(* Logix 5000 project; controller reports 1756-L63 rev 20.11; software revision 20.04; part 19 of 52 *)

        [1096].log_data[14].valid := 1, [1096].log_data[15].valid := 1, [1096].log_data[16].valid := 1, [1096].log_data[17].valid := 1, [1096].log_data[18].valid := 1, [1096].log_data[19].valid := 1, [1096].time.Year := 2023, [1096].time.Month := 1, [1096].time.Day := 13, [1096].time.Hour := 11, [1096].time.Minute := 44, [1096].time.Second := 59, [1097].log_data[0].min := 1.0, [1097].log_data[0].max := 1.0, [1097].log_data[0].total := 300.0, [1097].log_data[0].time := 300.0, [1097].log_data[0].minminute := 45, [1097].log_data[0].maxminute := 45, [1097].log_data[0].valid := 1, [1097].log_data[1].valid := 1, [1097].log_data[2].valid := 1, [1097].log_data[3].valid := 1, [1097].log_data[4].valid := 1, [1097].log_data[5].valid := 1, [1097].log_data[6].valid := 1, [1097].log_data[7].valid := 1, [1097].log_data[8].valid := 1, [1097].log_data[9].valid := 1, [1097].log_data[10].valid := 1, [1097].log_data[11].valid := 1, [1097].log_data[12].valid := 1, [1097].log_data[13].valid := 1, [1097].log_data[14].valid := 1, [1097].log_data[15].valid := 1, [1097].log_data[16].valid := 1, [1097].log_data[17].valid := 1, [1097].log_data[18].valid := 1, [1097].log_data[19].valid := 1, [1097].time.Year := 2023, [1097].time.Month := 1, [1097].time.Day := 13, [1097].time.Hour := 11, [1097].time.Minute := 49, [1097].time.Second := 59, [1098].log_data[0].min := 1.0, [1098].log_data[0].max := 1.0, [1098].log_data[0].total := 300.0, [1098].log_data[0].time := 300.0, [1098].log_data[0].minminute := 50, [1098].log_data[0].maxminute := 50, [1098].log_data[0].valid := 1, [1098].log_data[1].valid := 1, [1098].log_data[2].valid := 1, [1098].log_data[3].valid := 1, [1098].log_data[4].valid := 1, [1098].log_data[5].valid := 1, [1098].log_data[6].valid := 1, [1098].log_data[7].valid := 1, [1098].log_data[8].valid := 1, [1098].log_data[9].valid := 1,
        [1098].log_data[10].valid := 1, [1098].log_data[11].valid := 1, [1098].log_data[12].valid := 1, [1098].log_data[13].valid := 1, [1098].log_data[14].valid := 1, [1098].log_data[15].valid := 1, [1098].log_data[16].valid := 1, [1098].log_data[17].valid := 1, [1098].log_data[18].valid := 1, [1098].log_data[19].valid := 1, [1098].time.Year := 2023, [1098].time.Month := 1, [1098].time.Day := 13, [1098].time.Hour := 11, [1098].time.Minute := 54, [1098].time.Second := 59, [1099].log_data[0].min := 1.0, [1099].log_data[0].max := 1.0, [1099].log_data[0].total := 300.0, [1099].log_data[0].time := 300.0, [1099].log_data[0].minminute := 55, [1099].log_data[0].maxminute := 55, [1099].log_data[0].valid := 1, [1099].log_data[1].valid := 1, [1099].log_data[2].valid := 1, [1099].log_data[3].valid := 1, [1099].log_data[4].valid := 1, [1099].log_data[5].valid := 1, [1099].log_data[6].valid := 1, [1099].log_data[7].valid := 1, [1099].log_data[8].valid := 1, [1099].log_data[9].valid := 1, [1099].log_data[10].valid := 1, [1099].log_data[11].valid := 1, [1099].log_data[12].valid := 1, [1099].log_data[13].valid := 1, [1099].log_data[14].valid := 1, [1099].log_data[15].valid := 1, [1099].log_data[16].valid := 1, [1099].log_data[17].valid := 1, [1099].log_data[18].valid := 1, [1099].log_data[19].valid := 1, [1099].time.Year := 2023, [1099].time.Month := 1, [1099].time.Day := 13, [1099].time.Hour := 11, [1099].time.Minute := 59, [1099].time.Second := 59, [1100].log_data[0].min := 1.0, [1100].log_data[0].max := 1.0, [1100].log_data[0].total := 300.0, [1100].log_data[0].time := 300.0, [1100].log_data[0].valid := 1, [1100].log_data[1].valid := 1, [1100].log_data[2].valid := 1, [1100].log_data[3].valid := 1, [1100].log_data[4].valid := 1, [1100].log_data[5].valid := 1, [1100].log_data[6].valid := 1, [1100].log_data[7].valid := 1,
        [1100].log_data[8].valid := 1, [1100].log_data[9].valid := 1, [1100].log_data[10].valid := 1, [1100].log_data[11].valid := 1, [1100].log_data[12].valid := 1, [1100].log_data[13].valid := 1, [1100].log_data[14].valid := 1, [1100].log_data[15].valid := 1, [1100].log_data[16].valid := 1, [1100].log_data[17].valid := 1, [1100].log_data[18].valid := 1, [1100].log_data[19].valid := 1, [1100].time.Year := 2023, [1100].time.Month := 1, [1100].time.Day := 13, [1100].time.Hour := 12, [1100].time.Minute := 4, [1100].time.Second := 59, [1101].log_data[0].min := 1.0, [1101].log_data[0].max := 1.0, [1101].log_data[0].total := 300.0, [1101].log_data[0].time := 300.0, [1101].log_data[0].minminute := 5, [1101].log_data[0].maxminute := 5, [1101].log_data[0].valid := 1, [1101].log_data[1].valid := 1, [1101].log_data[2].valid := 1, [1101].log_data[3].valid := 1, [1101].log_data[4].valid := 1, [1101].log_data[5].valid := 1, [1101].log_data[6].valid := 1, [1101].log_data[7].valid := 1, [1101].log_data[8].valid := 1, [1101].log_data[9].valid := 1, [1101].log_data[10].valid := 1, [1101].log_data[11].valid := 1, [1101].log_data[12].valid := 1, [1101].log_data[13].valid := 1, [1101].log_data[14].valid := 1, [1101].log_data[15].valid := 1, [1101].log_data[16].valid := 1, [1101].log_data[17].valid := 1, [1101].log_data[18].valid := 1, [1101].log_data[19].valid := 1, [1101].time.Year := 2023, [1101].time.Month := 1, [1101].time.Day := 13, [1101].time.Hour := 12, [1101].time.Minute := 9, [1101].time.Second := 59, [1102].log_data[0].min := 1.0, [1102].log_data[0].max := 1.0, [1102].log_data[0].total := 300.0, [1102].log_data[0].time := 300.0, [1102].log_data[0].minminute := 10, [1102].log_data[0].maxminute := 10, [1102].log_data[0].valid := 1, [1102].log_data[1].valid := 1, [1102].log_data[2].valid := 1, [1102].log_data[3].valid := 1,
        [1102].log_data[4].valid := 1, [1102].log_data[5].valid := 1, [1102].log_data[6].valid := 1, [1102].log_data[7].valid := 1, [1102].log_data[8].valid := 1, [1102].log_data[9].valid := 1, [1102].log_data[10].valid := 1, [1102].log_data[11].valid := 1, [1102].log_data[12].valid := 1, [1102].log_data[13].valid := 1, [1102].log_data[14].valid := 1, [1102].log_data[15].valid := 1, [1102].log_data[16].valid := 1, [1102].log_data[17].valid := 1, [1102].log_data[18].valid := 1, [1102].log_data[19].valid := 1, [1102].time.Year := 2023, [1102].time.Month := 1, [1102].time.Day := 13, [1102].time.Hour := 12, [1102].time.Minute := 14, [1102].time.Second := 59, [1103].log_data[0].min := 1.0, [1103].log_data[0].max := 1.0, [1103].log_data[0].total := 300.0, [1103].log_data[0].time := 300.0, [1103].log_data[0].minminute := 15, [1103].log_data[0].maxminute := 15, [1103].log_data[0].valid := 1, [1103].log_data[1].valid := 1, [1103].log_data[2].valid := 1, [1103].log_data[3].valid := 1, [1103].log_data[4].valid := 1, [1103].log_data[5].valid := 1, [1103].log_data[6].valid := 1, [1103].log_data[7].valid := 1, [1103].log_data[8].valid := 1, [1103].log_data[9].valid := 1, [1103].log_data[10].valid := 1, [1103].log_data[11].valid := 1, [1103].log_data[12].valid := 1, [1103].log_data[13].valid := 1, [1103].log_data[14].valid := 1, [1103].log_data[15].valid := 1, [1103].log_data[16].valid := 1, [1103].log_data[17].valid := 1, [1103].log_data[18].valid := 1, [1103].log_data[19].valid := 1, [1103].time.Year := 2023, [1103].time.Month := 1, [1103].time.Day := 13, [1103].time.Hour := 12, [1103].time.Minute := 19, [1103].time.Second := 59, [1104].log_data[0].min := 1.0, [1104].log_data[0].max := 1.0, [1104].log_data[0].total := 300.0, [1104].log_data[0].time := 300.0, [1104].log_data[0].minminute := 20, [1104].log_data[0].maxminute := 20,
        [1104].log_data[0].valid := 1, [1104].log_data[1].valid := 1, [1104].log_data[2].valid := 1, [1104].log_data[3].valid := 1, [1104].log_data[4].valid := 1, [1104].log_data[5].valid := 1, [1104].log_data[6].valid := 1, [1104].log_data[7].valid := 1, [1104].log_data[8].valid := 1, [1104].log_data[9].valid := 1, [1104].log_data[10].valid := 1, [1104].log_data[11].valid := 1, [1104].log_data[12].valid := 1, [1104].log_data[13].valid := 1, [1104].log_data[14].valid := 1, [1104].log_data[15].valid := 1, [1104].log_data[16].valid := 1, [1104].log_data[17].valid := 1, [1104].log_data[18].valid := 1, [1104].log_data[19].valid := 1, [1104].time.Year := 2023, [1104].time.Month := 1, [1104].time.Day := 13, [1104].time.Hour := 12, [1104].time.Minute := 24, [1104].time.Second := 59, [1105].log_data[0].min := 1.0, [1105].log_data[0].max := 1.0, [1105].log_data[0].total := 300.0, [1105].log_data[0].time := 300.0, [1105].log_data[0].minminute := 25, [1105].log_data[0].maxminute := 25, [1105].log_data[0].valid := 1, [1105].log_data[1].valid := 1, [1105].log_data[2].valid := 1, [1105].log_data[3].valid := 1, [1105].log_data[4].valid := 1, [1105].log_data[5].valid := 1, [1105].log_data[6].valid := 1, [1105].log_data[7].valid := 1, [1105].log_data[8].valid := 1, [1105].log_data[9].valid := 1, [1105].log_data[10].valid := 1, [1105].log_data[11].valid := 1, [1105].log_data[12].valid := 1, [1105].log_data[13].valid := 1, [1105].log_data[14].valid := 1, [1105].log_data[15].valid := 1, [1105].log_data[16].valid := 1, [1105].log_data[17].valid := 1, [1105].log_data[18].valid := 1, [1105].log_data[19].valid := 1, [1105].time.Year := 2023, [1105].time.Month := 1, [1105].time.Day := 13, [1105].time.Hour := 12, [1105].time.Minute := 29, [1105].time.Second := 59, [1106].log_data[0].min := 1.0, [1106].log_data[0].max := 1.0,
        [1106].log_data[0].total := 300.0, [1106].log_data[0].time := 300.0, [1106].log_data[0].minminute := 30, [1106].log_data[0].maxminute := 30, [1106].log_data[0].valid := 1, [1106].log_data[1].valid := 1, [1106].log_data[2].valid := 1, [1106].log_data[3].valid := 1, [1106].log_data[4].valid := 1, [1106].log_data[5].valid := 1, [1106].log_data[6].valid := 1, [1106].log_data[7].valid := 1, [1106].log_data[8].valid := 1, [1106].log_data[9].valid := 1, [1106].log_data[10].valid := 1, [1106].log_data[11].valid := 1, [1106].log_data[12].valid := 1, [1106].log_data[13].valid := 1, [1106].log_data[14].valid := 1, [1106].log_data[15].valid := 1, [1106].log_data[16].valid := 1, [1106].log_data[17].valid := 1, [1106].log_data[18].valid := 1, [1106].log_data[19].valid := 1, [1106].time.Year := 2023, [1106].time.Month := 1, [1106].time.Day := 13, [1106].time.Hour := 12, [1106].time.Minute := 34, [1106].time.Second := 59, [1107].log_data[0].min := 1.0, [1107].log_data[0].max := 1.0, [1107].log_data[0].total := 300.0, [1107].log_data[0].time := 300.0, [1107].log_data[0].minminute := 35, [1107].log_data[0].maxminute := 35, [1107].log_data[0].valid := 1, [1107].log_data[1].valid := 1, [1107].log_data[2].valid := 1, [1107].log_data[3].valid := 1, [1107].log_data[4].valid := 1, [1107].log_data[5].valid := 1, [1107].log_data[6].valid := 1, [1107].log_data[7].valid := 1, [1107].log_data[8].valid := 1, [1107].log_data[9].valid := 1, [1107].log_data[10].valid := 1, [1107].log_data[11].valid := 1, [1107].log_data[12].valid := 1, [1107].log_data[13].valid := 1, [1107].log_data[14].valid := 1, [1107].log_data[15].valid := 1, [1107].log_data[16].valid := 1, [1107].log_data[17].valid := 1, [1107].log_data[18].valid := 1, [1107].log_data[19].valid := 1, [1107].time.Year := 2023, [1107].time.Month := 1, [1107].time.Day := 13, [1107].time.Hour := 12,
        [1107].time.Minute := 39, [1107].time.Second := 59, [1108].log_data[0].min := 1.0, [1108].log_data[0].max := 1.0, [1108].log_data[0].total := 300.0, [1108].log_data[0].time := 300.0, [1108].log_data[0].minminute := 40, [1108].log_data[0].maxminute := 40, [1108].log_data[0].valid := 1, [1108].log_data[1].valid := 1, [1108].log_data[2].valid := 1, [1108].log_data[3].valid := 1, [1108].log_data[4].valid := 1, [1108].log_data[5].valid := 1, [1108].log_data[6].valid := 1, [1108].log_data[7].valid := 1, [1108].log_data[8].valid := 1, [1108].log_data[9].valid := 1, [1108].log_data[10].valid := 1, [1108].log_data[11].valid := 1, [1108].log_data[12].valid := 1, [1108].log_data[13].valid := 1, [1108].log_data[14].valid := 1, [1108].log_data[15].valid := 1, [1108].log_data[16].valid := 1, [1108].log_data[17].valid := 1, [1108].log_data[18].valid := 1, [1108].log_data[19].valid := 1, [1108].time.Year := 2023, [1108].time.Month := 1, [1108].time.Day := 13, [1108].time.Hour := 12, [1108].time.Minute := 44, [1108].time.Second := 59, [1109].log_data[0].min := 1.0, [1109].log_data[0].max := 1.0, [1109].log_data[0].total := 300.0, [1109].log_data[0].time := 300.0, [1109].log_data[0].minminute := 45, [1109].log_data[0].maxminute := 45, [1109].log_data[0].valid := 1, [1109].log_data[1].valid := 1, [1109].log_data[2].valid := 1, [1109].log_data[3].valid := 1, [1109].log_data[4].valid := 1, [1109].log_data[5].valid := 1, [1109].log_data[6].valid := 1, [1109].log_data[7].valid := 1, [1109].log_data[8].valid := 1, [1109].log_data[9].valid := 1, [1109].log_data[10].valid := 1, [1109].log_data[11].valid := 1, [1109].log_data[12].valid := 1, [1109].log_data[13].valid := 1, [1109].log_data[14].valid := 1, [1109].log_data[15].valid := 1, [1109].log_data[16].valid := 1, [1109].log_data[17].valid := 1, [1109].log_data[18].valid := 1, [1109].log_data[19].valid := 1,
        [1109].time.Year := 2023, [1109].time.Month := 1, [1109].time.Day := 13, [1109].time.Hour := 12, [1109].time.Minute := 49, [1109].time.Second := 59, [1110].log_data[0].min := 1.0, [1110].log_data[0].max := 1.0, [1110].log_data[0].total := 300.0, [1110].log_data[0].time := 300.0, [1110].log_data[0].minminute := 50, [1110].log_data[0].maxminute := 50, [1110].log_data[0].valid := 1, [1110].log_data[1].valid := 1, [1110].log_data[2].valid := 1, [1110].log_data[3].valid := 1, [1110].log_data[4].valid := 1, [1110].log_data[5].valid := 1, [1110].log_data[6].valid := 1, [1110].log_data[7].valid := 1, [1110].log_data[8].valid := 1, [1110].log_data[9].valid := 1, [1110].log_data[10].valid := 1, [1110].log_data[11].valid := 1, [1110].log_data[12].valid := 1, [1110].log_data[13].valid := 1, [1110].log_data[14].valid := 1, [1110].log_data[15].valid := 1, [1110].log_data[16].valid := 1, [1110].log_data[17].valid := 1, [1110].log_data[18].valid := 1, [1110].log_data[19].valid := 1, [1110].time.Year := 2023, [1110].time.Month := 1, [1110].time.Day := 13, [1110].time.Hour := 12, [1110].time.Minute := 54, [1110].time.Second := 59, [1111].log_data[0].min := 1.0, [1111].log_data[0].max := 1.0, [1111].log_data[0].total := 300.0, [1111].log_data[0].time := 300.0, [1111].log_data[0].minminute := 55, [1111].log_data[0].maxminute := 55, [1111].log_data[0].valid := 1, [1111].log_data[1].valid := 1, [1111].log_data[2].valid := 1, [1111].log_data[3].valid := 1, [1111].log_data[4].valid := 1, [1111].log_data[5].valid := 1, [1111].log_data[6].valid := 1, [1111].log_data[7].valid := 1, [1111].log_data[8].valid := 1, [1111].log_data[9].valid := 1, [1111].log_data[10].valid := 1, [1111].log_data[11].valid := 1, [1111].log_data[12].valid := 1, [1111].log_data[13].valid := 1, [1111].log_data[14].valid := 1, [1111].log_data[15].valid := 1,
        [1111].log_data[16].valid := 1, [1111].log_data[17].valid := 1, [1111].log_data[18].valid := 1, [1111].log_data[19].valid := 1, [1111].time.Year := 2023, [1111].time.Month := 1, [1111].time.Day := 13, [1111].time.Hour := 12, [1111].time.Minute := 59, [1111].time.Second := 59, [1112].log_data[0].min := 1.0, [1112].log_data[0].max := 1.0, [1112].log_data[0].total := 299.5, [1112].log_data[0].time := 299.5, [1112].log_data[0].valid := 1, [1112].log_data[1].valid := 1, [1112].log_data[2].valid := 1, [1112].log_data[3].valid := 1, [1112].log_data[4].valid := 1, [1112].log_data[5].valid := 1, [1112].log_data[6].valid := 1, [1112].log_data[7].valid := 1, [1112].log_data[8].valid := 1, [1112].log_data[9].valid := 1, [1112].log_data[10].valid := 1, [1112].log_data[11].valid := 1, [1112].log_data[12].valid := 1, [1112].log_data[13].valid := 1, [1112].log_data[14].valid := 1, [1112].log_data[15].valid := 1, [1112].log_data[16].valid := 1, [1112].log_data[17].valid := 1, [1112].log_data[18].valid := 1, [1112].log_data[19].valid := 1, [1112].time.Year := 2023, [1112].time.Month := 1, [1112].time.Day := 13, [1112].time.Hour := 13, [1112].time.Minute := 4, [1112].time.Second := 59, [1113].log_data[0].min := 1.0, [1113].log_data[0].max := 1.0, [1113].log_data[0].total := 300.0, [1113].log_data[0].time := 300.0, [1113].log_data[0].minminute := 5, [1113].log_data[0].maxminute := 5, [1113].log_data[0].valid := 1, [1113].log_data[1].valid := 1, [1113].log_data[2].valid := 1, [1113].log_data[3].valid := 1, [1113].log_data[4].valid := 1, [1113].log_data[5].valid := 1, [1113].log_data[6].valid := 1, [1113].log_data[7].valid := 1, [1113].log_data[8].valid := 1, [1113].log_data[9].valid := 1, [1113].log_data[10].valid := 1, [1113].log_data[11].valid := 1, [1113].log_data[12].valid := 1, [1113].log_data[13].valid := 1,
        [1113].log_data[14].valid := 1, [1113].log_data[15].valid := 1, [1113].log_data[16].valid := 1, [1113].log_data[17].valid := 1, [1113].log_data[18].valid := 1, [1113].log_data[19].valid := 1, [1113].time.Year := 2023, [1113].time.Month := 1, [1113].time.Day := 13, [1113].time.Hour := 13, [1113].time.Minute := 9, [1113].time.Second := 59, [1114].log_data[0].min := 1.0, [1114].log_data[0].max := 1.0, [1114].log_data[0].total := 300.0, [1114].log_data[0].time := 300.0, [1114].log_data[0].minminute := 10, [1114].log_data[0].maxminute := 10, [1114].log_data[0].valid := 1, [1114].log_data[1].valid := 1, [1114].log_data[2].valid := 1, [1114].log_data[3].valid := 1, [1114].log_data[4].valid := 1, [1114].log_data[5].valid := 1, [1114].log_data[6].valid := 1, [1114].log_data[7].valid := 1, [1114].log_data[8].valid := 1, [1114].log_data[9].valid := 1, [1114].log_data[10].valid := 1, [1114].log_data[11].valid := 1, [1114].log_data[12].valid := 1, [1114].log_data[13].valid := 1, [1114].log_data[14].valid := 1, [1114].log_data[15].valid := 1, [1114].log_data[16].valid := 1, [1114].log_data[17].valid := 1, [1114].log_data[18].valid := 1, [1114].log_data[19].valid := 1, [1114].time.Year := 2023, [1114].time.Month := 1, [1114].time.Day := 13, [1114].time.Hour := 13, [1114].time.Minute := 14, [1114].time.Second := 59, [1115].log_data[0].min := 1.0, [1115].log_data[0].max := 1.0, [1115].log_data[0].total := 300.0, [1115].log_data[0].time := 300.0, [1115].log_data[0].minminute := 15, [1115].log_data[0].maxminute := 15, [1115].log_data[0].valid := 1, [1115].log_data[1].valid := 1, [1115].log_data[2].valid := 1, [1115].log_data[3].valid := 1, [1115].log_data[4].valid := 1, [1115].log_data[5].valid := 1, [1115].log_data[6].valid := 1, [1115].log_data[7].valid := 1, [1115].log_data[8].valid := 1, [1115].log_data[9].valid := 1,
        [1115].log_data[10].valid := 1, [1115].log_data[11].valid := 1, [1115].log_data[12].valid := 1, [1115].log_data[13].valid := 1, [1115].log_data[14].valid := 1, [1115].log_data[15].valid := 1, [1115].log_data[16].valid := 1, [1115].log_data[17].valid := 1, [1115].log_data[18].valid := 1, [1115].log_data[19].valid := 1, [1115].time.Year := 2023, [1115].time.Month := 1, [1115].time.Day := 13, [1115].time.Hour := 13, [1115].time.Minute := 19, [1115].time.Second := 59, [1116].log_data[0].min := 1.0, [1116].log_data[0].max := 1.0, [1116].log_data[0].total := 300.0, [1116].log_data[0].time := 300.0, [1116].log_data[0].minminute := 20, [1116].log_data[0].maxminute := 20, [1116].log_data[0].valid := 1, [1116].log_data[1].valid := 1, [1116].log_data[2].valid := 1, [1116].log_data[3].valid := 1, [1116].log_data[4].valid := 1, [1116].log_data[5].valid := 1, [1116].log_data[6].valid := 1, [1116].log_data[7].valid := 1, [1116].log_data[8].valid := 1, [1116].log_data[9].valid := 1, [1116].log_data[10].valid := 1, [1116].log_data[11].valid := 1, [1116].log_data[12].valid := 1, [1116].log_data[13].valid := 1, [1116].log_data[14].valid := 1, [1116].log_data[15].valid := 1, [1116].log_data[16].valid := 1, [1116].log_data[17].valid := 1, [1116].log_data[18].valid := 1, [1116].log_data[19].valid := 1, [1116].time.Year := 2023, [1116].time.Month := 1, [1116].time.Day := 13, [1116].time.Hour := 13, [1116].time.Minute := 24, [1116].time.Second := 59, [1117].log_data[0].min := 1.0, [1117].log_data[0].max := 1.0, [1117].log_data[0].total := 300.0, [1117].log_data[0].time := 300.0, [1117].log_data[0].minminute := 25, [1117].log_data[0].maxminute := 25, [1117].log_data[0].valid := 1, [1117].log_data[1].valid := 1, [1117].log_data[2].valid := 1, [1117].log_data[3].valid := 1, [1117].log_data[4].valid := 1, [1117].log_data[5].valid := 1,
        [1117].log_data[6].valid := 1, [1117].log_data[7].valid := 1, [1117].log_data[8].valid := 1, [1117].log_data[9].valid := 1, [1117].log_data[10].valid := 1, [1117].log_data[11].valid := 1, [1117].log_data[12].valid := 1, [1117].log_data[13].valid := 1, [1117].log_data[14].valid := 1, [1117].log_data[15].valid := 1, [1117].log_data[16].valid := 1, [1117].log_data[17].valid := 1, [1117].log_data[18].valid := 1, [1117].log_data[19].valid := 1, [1117].time.Year := 2023, [1117].time.Month := 1, [1117].time.Day := 13, [1117].time.Hour := 13, [1117].time.Minute := 29, [1117].time.Second := 59, [1118].log_data[0].min := 1.0, [1118].log_data[0].max := 1.0, [1118].log_data[0].total := 300.0, [1118].log_data[0].time := 300.0, [1118].log_data[0].minminute := 30, [1118].log_data[0].maxminute := 30, [1118].log_data[0].valid := 1, [1118].log_data[1].valid := 1, [1118].log_data[2].valid := 1, [1118].log_data[3].valid := 1, [1118].log_data[4].valid := 1, [1118].log_data[5].valid := 1, [1118].log_data[6].valid := 1, [1118].log_data[7].valid := 1, [1118].log_data[8].valid := 1, [1118].log_data[9].valid := 1, [1118].log_data[10].valid := 1, [1118].log_data[11].valid := 1, [1118].log_data[12].valid := 1, [1118].log_data[13].valid := 1, [1118].log_data[14].valid := 1, [1118].log_data[15].valid := 1, [1118].log_data[16].valid := 1, [1118].log_data[17].valid := 1, [1118].log_data[18].valid := 1, [1118].log_data[19].valid := 1, [1118].time.Year := 2023, [1118].time.Month := 1, [1118].time.Day := 13, [1118].time.Hour := 13, [1118].time.Minute := 34, [1118].time.Second := 59, [1119].log_data[0].min := 1.0, [1119].log_data[0].max := 1.0, [1119].log_data[0].total := 300.0, [1119].log_data[0].time := 300.0, [1119].log_data[0].minminute := 35, [1119].log_data[0].maxminute := 35, [1119].log_data[0].valid := 1, [1119].log_data[1].valid := 1,
        [1119].log_data[2].valid := 1, [1119].log_data[3].valid := 1, [1119].log_data[4].valid := 1, [1119].log_data[5].valid := 1, [1119].log_data[6].valid := 1, [1119].log_data[7].valid := 1, [1119].log_data[8].valid := 1, [1119].log_data[9].valid := 1, [1119].log_data[10].valid := 1, [1119].log_data[11].valid := 1, [1119].log_data[12].valid := 1, [1119].log_data[13].valid := 1, [1119].log_data[14].valid := 1, [1119].log_data[15].valid := 1, [1119].log_data[16].valid := 1, [1119].log_data[17].valid := 1, [1119].log_data[18].valid := 1, [1119].log_data[19].valid := 1, [1119].time.Year := 2023, [1119].time.Month := 1, [1119].time.Day := 13, [1119].time.Hour := 13, [1119].time.Minute := 39, [1119].time.Second := 59, [1120].log_data[0].min := 1.0, [1120].log_data[0].max := 1.0, [1120].log_data[0].total := 300.0, [1120].log_data[0].time := 300.0, [1120].log_data[0].minminute := 40, [1120].log_data[0].maxminute := 40, [1120].log_data[0].valid := 1, [1120].log_data[1].valid := 1, [1120].log_data[2].valid := 1, [1120].log_data[3].valid := 1, [1120].log_data[4].valid := 1, [1120].log_data[5].valid := 1, [1120].log_data[6].valid := 1, [1120].log_data[7].valid := 1, [1120].log_data[8].valid := 1, [1120].log_data[9].valid := 1, [1120].log_data[10].valid := 1, [1120].log_data[11].valid := 1, [1120].log_data[12].valid := 1, [1120].log_data[13].valid := 1, [1120].log_data[14].valid := 1, [1120].log_data[15].valid := 1, [1120].log_data[16].valid := 1, [1120].log_data[17].valid := 1, [1120].log_data[18].valid := 1, [1120].log_data[19].valid := 1, [1120].time.Year := 2023, [1120].time.Month := 1, [1120].time.Day := 13, [1120].time.Hour := 13, [1120].time.Minute := 44, [1120].time.Second := 59, [1121].log_data[0].min := 1.0, [1121].log_data[0].max := 1.0, [1121].log_data[0].total := 300.0, [1121].log_data[0].time := 300.0,
        [1121].log_data[0].minminute := 45, [1121].log_data[0].maxminute := 45, [1121].log_data[0].valid := 1, [1121].log_data[1].valid := 1, [1121].log_data[2].valid := 1, [1121].log_data[3].valid := 1, [1121].log_data[4].valid := 1, [1121].log_data[5].valid := 1, [1121].log_data[6].valid := 1, [1121].log_data[7].valid := 1, [1121].log_data[8].valid := 1, [1121].log_data[9].valid := 1, [1121].log_data[10].valid := 1, [1121].log_data[11].valid := 1, [1121].log_data[12].valid := 1, [1121].log_data[13].valid := 1, [1121].log_data[14].valid := 1, [1121].log_data[15].valid := 1, [1121].log_data[16].valid := 1, [1121].log_data[17].valid := 1, [1121].log_data[18].valid := 1, [1121].log_data[19].valid := 1, [1121].time.Year := 2023, [1121].time.Month := 1, [1121].time.Day := 13, [1121].time.Hour := 13, [1121].time.Minute := 49, [1121].time.Second := 59, [1122].log_data[0].min := 1.0, [1122].log_data[0].max := 1.0, [1122].log_data[0].total := 300.0, [1122].log_data[0].time := 300.0, [1122].log_data[0].minminute := 50, [1122].log_data[0].maxminute := 50, [1122].log_data[0].valid := 1, [1122].log_data[1].valid := 1, [1122].log_data[2].valid := 1, [1122].log_data[3].valid := 1, [1122].log_data[4].valid := 1, [1122].log_data[5].valid := 1, [1122].log_data[6].valid := 1, [1122].log_data[7].valid := 1, [1122].log_data[8].valid := 1, [1122].log_data[9].valid := 1, [1122].log_data[10].valid := 1, [1122].log_data[11].valid := 1, [1122].log_data[12].valid := 1, [1122].log_data[13].valid := 1, [1122].log_data[14].valid := 1, [1122].log_data[15].valid := 1, [1122].log_data[16].valid := 1, [1122].log_data[17].valid := 1, [1122].log_data[18].valid := 1, [1122].log_data[19].valid := 1, [1122].time.Year := 2023, [1122].time.Month := 1, [1122].time.Day := 13, [1122].time.Hour := 13, [1122].time.Minute := 54, [1122].time.Second := 59,
        [1123].log_data[0].min := 1.0, [1123].log_data[0].max := 1.0, [1123].log_data[0].total := 300.0, [1123].log_data[0].time := 300.0, [1123].log_data[0].minminute := 55, [1123].log_data[0].maxminute := 55, [1123].log_data[0].valid := 1, [1123].log_data[1].valid := 1, [1123].log_data[2].valid := 1, [1123].log_data[3].valid := 1, [1123].log_data[4].valid := 1, [1123].log_data[5].valid := 1, [1123].log_data[6].valid := 1, [1123].log_data[7].valid := 1, [1123].log_data[8].valid := 1, [1123].log_data[9].valid := 1, [1123].log_data[10].valid := 1, [1123].log_data[11].valid := 1, [1123].log_data[12].valid := 1, [1123].log_data[13].valid := 1, [1123].log_data[14].valid := 1, [1123].log_data[15].valid := 1, [1123].log_data[16].valid := 1, [1123].log_data[17].valid := 1, [1123].log_data[18].valid := 1, [1123].log_data[19].valid := 1, [1123].time.Year := 2023, [1123].time.Month := 1, [1123].time.Day := 13, [1123].time.Hour := 13, [1123].time.Minute := 59, [1123].time.Second := 59, [1124].log_data[0].min := 1.0, [1124].log_data[0].max := 1.0, [1124].log_data[0].total := 300.0, [1124].log_data[0].time := 300.0, [1124].log_data[0].valid := 1, [1124].log_data[1].valid := 1, [1124].log_data[2].valid := 1, [1124].log_data[3].valid := 1, [1124].log_data[4].valid := 1, [1124].log_data[5].valid := 1, [1124].log_data[6].valid := 1, [1124].log_data[7].valid := 1, [1124].log_data[8].valid := 1, [1124].log_data[9].valid := 1, [1124].log_data[10].valid := 1, [1124].log_data[11].valid := 1, [1124].log_data[12].valid := 1, [1124].log_data[13].valid := 1, [1124].log_data[14].valid := 1, [1124].log_data[15].valid := 1, [1124].log_data[16].valid := 1, [1124].log_data[17].valid := 1, [1124].log_data[18].valid := 1, [1124].log_data[19].valid := 1, [1124].time.Year := 2023, [1124].time.Month := 1, [1124].time.Day := 13, [1124].time.Hour := 14,
        [1124].time.Minute := 4, [1124].time.Second := 59, [1125].log_data[0].min := 1.0, [1125].log_data[0].max := 1.0, [1125].log_data[0].total := 300.0, [1125].log_data[0].time := 300.0, [1125].log_data[0].minminute := 5, [1125].log_data[0].maxminute := 5, [1125].log_data[0].valid := 1, [1125].log_data[1].valid := 1, [1125].log_data[2].valid := 1, [1125].log_data[3].valid := 1, [1125].log_data[4].valid := 1, [1125].log_data[5].valid := 1, [1125].log_data[6].valid := 1, [1125].log_data[7].valid := 1, [1125].log_data[8].valid := 1, [1125].log_data[9].valid := 1, [1125].log_data[10].valid := 1, [1125].log_data[11].valid := 1, [1125].log_data[12].valid := 1, [1125].log_data[13].valid := 1, [1125].log_data[14].valid := 1, [1125].log_data[15].valid := 1, [1125].log_data[16].valid := 1, [1125].log_data[17].valid := 1, [1125].log_data[18].valid := 1, [1125].log_data[19].valid := 1, [1125].time.Year := 2023, [1125].time.Month := 1, [1125].time.Day := 13, [1125].time.Hour := 14, [1125].time.Minute := 9, [1125].time.Second := 59, [1126].log_data[0].min := 1.0, [1126].log_data[0].max := 1.0, [1126].log_data[0].total := 300.0, [1126].log_data[0].time := 300.0, [1126].log_data[0].minminute := 10, [1126].log_data[0].maxminute := 10, [1126].log_data[0].valid := 1, [1126].log_data[1].valid := 1, [1126].log_data[2].valid := 1, [1126].log_data[3].valid := 1, [1126].log_data[4].valid := 1, [1126].log_data[5].valid := 1, [1126].log_data[6].valid := 1, [1126].log_data[7].valid := 1, [1126].log_data[8].valid := 1, [1126].log_data[9].valid := 1, [1126].log_data[10].valid := 1, [1126].log_data[11].valid := 1, [1126].log_data[12].valid := 1, [1126].log_data[13].valid := 1, [1126].log_data[14].valid := 1, [1126].log_data[15].valid := 1, [1126].log_data[16].valid := 1, [1126].log_data[17].valid := 1, [1126].log_data[18].valid := 1, [1126].log_data[19].valid := 1,
        [1126].time.Year := 2023, [1126].time.Month := 1, [1126].time.Day := 13, [1126].time.Hour := 14, [1126].time.Minute := 14, [1126].time.Second := 59, [1127].log_data[0].min := 1.0, [1127].log_data[0].max := 1.0, [1127].log_data[0].total := 300.0, [1127].log_data[0].time := 300.0, [1127].log_data[0].minminute := 15, [1127].log_data[0].maxminute := 15, [1127].log_data[0].valid := 1, [1127].log_data[1].valid := 1, [1127].log_data[2].valid := 1, [1127].log_data[3].valid := 1, [1127].log_data[4].valid := 1, [1127].log_data[5].valid := 1, [1127].log_data[6].valid := 1, [1127].log_data[7].valid := 1, [1127].log_data[8].valid := 1, [1127].log_data[9].valid := 1, [1127].log_data[10].valid := 1, [1127].log_data[11].valid := 1, [1127].log_data[12].valid := 1, [1127].log_data[13].valid := 1, [1127].log_data[14].valid := 1, [1127].log_data[15].valid := 1, [1127].log_data[16].valid := 1, [1127].log_data[17].valid := 1, [1127].log_data[18].valid := 1, [1127].log_data[19].valid := 1, [1127].time.Year := 2023, [1127].time.Month := 1, [1127].time.Day := 13, [1127].time.Hour := 14, [1127].time.Minute := 19, [1127].time.Second := 59, [1128].log_data[0].min := 1.0, [1128].log_data[0].max := 1.0, [1128].log_data[0].total := 300.0, [1128].log_data[0].time := 300.0, [1128].log_data[0].minminute := 20, [1128].log_data[0].maxminute := 20, [1128].log_data[0].valid := 1, [1128].log_data[1].valid := 1, [1128].log_data[2].valid := 1, [1128].log_data[3].valid := 1, [1128].log_data[4].valid := 1, [1128].log_data[5].valid := 1, [1128].log_data[6].valid := 1, [1128].log_data[7].valid := 1, [1128].log_data[8].valid := 1, [1128].log_data[9].valid := 1, [1128].log_data[10].valid := 1, [1128].log_data[11].valid := 1, [1128].log_data[12].valid := 1, [1128].log_data[13].valid := 1, [1128].log_data[14].valid := 1, [1128].log_data[15].valid := 1,
        [1128].log_data[16].valid := 1, [1128].log_data[17].valid := 1, [1128].log_data[18].valid := 1, [1128].log_data[19].valid := 1, [1128].time.Year := 2023, [1128].time.Month := 1, [1128].time.Day := 13, [1128].time.Hour := 14, [1128].time.Minute := 24, [1128].time.Second := 59, [1129].log_data[0].min := 1.0, [1129].log_data[0].max := 1.0, [1129].log_data[0].total := 300.0, [1129].log_data[0].time := 300.0, [1129].log_data[0].minminute := 25, [1129].log_data[0].maxminute := 25, [1129].log_data[0].valid := 1, [1129].log_data[1].valid := 1, [1129].log_data[2].valid := 1, [1129].log_data[3].valid := 1, [1129].log_data[4].valid := 1, [1129].log_data[5].valid := 1, [1129].log_data[6].valid := 1, [1129].log_data[7].valid := 1, [1129].log_data[8].valid := 1, [1129].log_data[9].valid := 1, [1129].log_data[10].valid := 1, [1129].log_data[11].valid := 1, [1129].log_data[12].valid := 1, [1129].log_data[13].valid := 1, [1129].log_data[14].valid := 1, [1129].log_data[15].valid := 1, [1129].log_data[16].valid := 1, [1129].log_data[17].valid := 1, [1129].log_data[18].valid := 1, [1129].log_data[19].valid := 1, [1129].time.Year := 2023, [1129].time.Month := 1, [1129].time.Day := 13, [1129].time.Hour := 14, [1129].time.Minute := 29, [1129].time.Second := 59, [1130].log_data[0].min := 1.0, [1130].log_data[0].max := 1.0, [1130].log_data[0].total := 300.0, [1130].log_data[0].time := 300.0, [1130].log_data[0].minminute := 30, [1130].log_data[0].maxminute := 30, [1130].log_data[0].valid := 1, [1130].log_data[1].valid := 1, [1130].log_data[2].valid := 1, [1130].log_data[3].valid := 1, [1130].log_data[4].valid := 1, [1130].log_data[5].valid := 1, [1130].log_data[6].valid := 1, [1130].log_data[7].valid := 1, [1130].log_data[8].valid := 1, [1130].log_data[9].valid := 1, [1130].log_data[10].valid := 1, [1130].log_data[11].valid := 1,
        [1130].log_data[12].valid := 1, [1130].log_data[13].valid := 1, [1130].log_data[14].valid := 1, [1130].log_data[15].valid := 1, [1130].log_data[16].valid := 1, [1130].log_data[17].valid := 1, [1130].log_data[18].valid := 1, [1130].log_data[19].valid := 1, [1130].time.Year := 2023, [1130].time.Month := 1, [1130].time.Day := 13, [1130].time.Hour := 14, [1130].time.Minute := 34, [1130].time.Second := 59, [1131].log_data[0].min := 1.0, [1131].log_data[0].max := 1.0, [1131].log_data[0].total := 300.0, [1131].log_data[0].time := 300.0, [1131].log_data[0].minminute := 35, [1131].log_data[0].maxminute := 35, [1131].log_data[0].valid := 1, [1131].log_data[1].valid := 1, [1131].log_data[2].valid := 1, [1131].log_data[3].valid := 1, [1131].log_data[4].valid := 1, [1131].log_data[5].valid := 1, [1131].log_data[6].valid := 1, [1131].log_data[7].valid := 1, [1131].log_data[8].valid := 1, [1131].log_data[9].valid := 1, [1131].log_data[10].valid := 1, [1131].log_data[11].valid := 1, [1131].log_data[12].valid := 1, [1131].log_data[13].valid := 1, [1131].log_data[14].valid := 1, [1131].log_data[15].valid := 1, [1131].log_data[16].valid := 1, [1131].log_data[17].valid := 1, [1131].log_data[18].valid := 1, [1131].log_data[19].valid := 1, [1131].time.Year := 2023, [1131].time.Month := 1, [1131].time.Day := 13, [1131].time.Hour := 14, [1131].time.Minute := 39, [1131].time.Second := 59, [1132].log_data[0].min := 1.0, [1132].log_data[0].max := 1.0, [1132].log_data[0].total := 300.0, [1132].log_data[0].time := 300.0, [1132].log_data[0].minminute := 40, [1132].log_data[0].maxminute := 40, [1132].log_data[0].valid := 1, [1132].log_data[1].valid := 1, [1132].log_data[2].valid := 1, [1132].log_data[3].valid := 1, [1132].log_data[4].valid := 1, [1132].log_data[5].valid := 1, [1132].log_data[6].valid := 1, [1132].log_data[7].valid := 1,
        [1132].log_data[8].valid := 1, [1132].log_data[9].valid := 1, [1132].log_data[10].valid := 1, [1132].log_data[11].valid := 1, [1132].log_data[12].valid := 1, [1132].log_data[13].valid := 1, [1132].log_data[14].valid := 1, [1132].log_data[15].valid := 1, [1132].log_data[16].valid := 1, [1132].log_data[17].valid := 1, [1132].log_data[18].valid := 1, [1132].log_data[19].valid := 1, [1132].time.Year := 2023, [1132].time.Month := 1, [1132].time.Day := 13, [1132].time.Hour := 14, [1132].time.Minute := 44, [1132].time.Second := 59, [1133].log_data[0].min := 1.0, [1133].log_data[0].max := 1.0, [1133].log_data[0].total := 300.0, [1133].log_data[0].time := 300.0, [1133].log_data[0].minminute := 45, [1133].log_data[0].maxminute := 45, [1133].log_data[0].valid := 1, [1133].log_data[1].valid := 1, [1133].log_data[2].valid := 1, [1133].log_data[3].valid := 1, [1133].log_data[4].valid := 1, [1133].log_data[5].valid := 1, [1133].log_data[6].valid := 1, [1133].log_data[7].valid := 1, [1133].log_data[8].valid := 1, [1133].log_data[9].valid := 1, [1133].log_data[10].valid := 1, [1133].log_data[11].valid := 1, [1133].log_data[12].valid := 1, [1133].log_data[13].valid := 1, [1133].log_data[14].valid := 1, [1133].log_data[15].valid := 1, [1133].log_data[16].valid := 1, [1133].log_data[17].valid := 1, [1133].log_data[18].valid := 1, [1133].log_data[19].valid := 1, [1133].time.Year := 2023, [1133].time.Month := 1, [1133].time.Day := 13, [1133].time.Hour := 14, [1133].time.Minute := 49, [1133].time.Second := 59, [1134].log_data[0].min := 1.0, [1134].log_data[0].max := 1.0, [1134].log_data[0].total := 300.0, [1134].log_data[0].time := 300.0, [1134].log_data[0].minminute := 50, [1134].log_data[0].maxminute := 50, [1134].log_data[0].valid := 1, [1134].log_data[1].valid := 1, [1134].log_data[2].valid := 1, [1134].log_data[3].valid := 1,
        [1134].log_data[4].valid := 1, [1134].log_data[5].valid := 1, [1134].log_data[6].valid := 1, [1134].log_data[7].valid := 1, [1134].log_data[8].valid := 1, [1134].log_data[9].valid := 1, [1134].log_data[10].valid := 1, [1134].log_data[11].valid := 1, [1134].log_data[12].valid := 1, [1134].log_data[13].valid := 1, [1134].log_data[14].valid := 1, [1134].log_data[15].valid := 1, [1134].log_data[16].valid := 1, [1134].log_data[17].valid := 1, [1134].log_data[18].valid := 1, [1134].log_data[19].valid := 1, [1134].time.Year := 2023, [1134].time.Month := 1, [1134].time.Day := 13, [1134].time.Hour := 14, [1134].time.Minute := 54, [1134].time.Second := 59, [1135].log_data[0].min := 1.0, [1135].log_data[0].max := 1.0, [1135].log_data[0].total := 300.0, [1135].log_data[0].time := 300.0, [1135].log_data[0].minminute := 55, [1135].log_data[0].maxminute := 55, [1135].log_data[0].valid := 1, [1135].log_data[1].valid := 1, [1135].log_data[2].valid := 1, [1135].log_data[3].valid := 1, [1135].log_data[4].valid := 1, [1135].log_data[5].valid := 1, [1135].log_data[6].valid := 1, [1135].log_data[7].valid := 1, [1135].log_data[8].valid := 1, [1135].log_data[9].valid := 1, [1135].log_data[10].valid := 1, [1135].log_data[11].valid := 1, [1135].log_data[12].valid := 1, [1135].log_data[13].valid := 1, [1135].log_data[14].valid := 1, [1135].log_data[15].valid := 1, [1135].log_data[16].valid := 1, [1135].log_data[17].valid := 1, [1135].log_data[18].valid := 1, [1135].log_data[19].valid := 1, [1135].time.Year := 2023, [1135].time.Month := 1, [1135].time.Day := 13, [1135].time.Hour := 14, [1135].time.Minute := 59, [1135].time.Second := 59, [1136].log_data[0].min := 1.0, [1136].log_data[0].max := 1.0, [1136].log_data[0].total := 300.0, [1136].log_data[0].time := 300.0, [1136].log_data[0].valid := 1, [1136].log_data[1].valid := 1,
        [1136].log_data[2].valid := 1, [1136].log_data[3].valid := 1, [1136].log_data[4].valid := 1, [1136].log_data[5].valid := 1, [1136].log_data[6].valid := 1, [1136].log_data[7].valid := 1, [1136].log_data[8].valid := 1, [1136].log_data[9].valid := 1, [1136].log_data[10].valid := 1, [1136].log_data[11].valid := 1, [1136].log_data[12].valid := 1, [1136].log_data[13].valid := 1, [1136].log_data[14].valid := 1, [1136].log_data[15].valid := 1, [1136].log_data[16].valid := 1, [1136].log_data[17].valid := 1, [1136].log_data[18].valid := 1, [1136].log_data[19].valid := 1, [1136].time.Year := 2023, [1136].time.Month := 1, [1136].time.Day := 13, [1136].time.Hour := 15, [1136].time.Minute := 4, [1136].time.Second := 59, [1137].log_data[0].min := 1.0, [1137].log_data[0].max := 1.0, [1137].log_data[0].total := 300.0, [1137].log_data[0].time := 300.0, [1137].log_data[0].minminute := 5, [1137].log_data[0].maxminute := 5, [1137].log_data[0].valid := 1, [1137].log_data[1].valid := 1, [1137].log_data[2].valid := 1, [1137].log_data[3].valid := 1, [1137].log_data[4].valid := 1, [1137].log_data[5].valid := 1, [1137].log_data[6].valid := 1, [1137].log_data[7].valid := 1, [1137].log_data[8].valid := 1, [1137].log_data[9].valid := 1, [1137].log_data[10].valid := 1, [1137].log_data[11].valid := 1, [1137].log_data[12].valid := 1, [1137].log_data[13].valid := 1, [1137].log_data[14].valid := 1, [1137].log_data[15].valid := 1, [1137].log_data[16].valid := 1, [1137].log_data[17].valid := 1, [1137].log_data[18].valid := 1, [1137].log_data[19].valid := 1, [1137].time.Year := 2023, [1137].time.Month := 1, [1137].time.Day := 13, [1137].time.Hour := 15, [1137].time.Minute := 9, [1137].time.Second := 59, [1138].log_data[0].min := 1.0, [1138].log_data[0].max := 1.0, [1138].log_data[0].total := 300.0, [1138].log_data[0].time := 300.0,
        [1138].log_data[0].minminute := 10, [1138].log_data[0].maxminute := 10, [1138].log_data[0].valid := 1, [1138].log_data[1].valid := 1, [1138].log_data[2].valid := 1, [1138].log_data[3].valid := 1, [1138].log_data[4].valid := 1, [1138].log_data[5].valid := 1, [1138].log_data[6].valid := 1, [1138].log_data[7].valid := 1, [1138].log_data[8].valid := 1, [1138].log_data[9].valid := 1, [1138].log_data[10].valid := 1, [1138].log_data[11].valid := 1, [1138].log_data[12].valid := 1, [1138].log_data[13].valid := 1, [1138].log_data[14].valid := 1, [1138].log_data[15].valid := 1, [1138].log_data[16].valid := 1, [1138].log_data[17].valid := 1, [1138].log_data[18].valid := 1, [1138].log_data[19].valid := 1, [1138].time.Year := 2023, [1138].time.Month := 1, [1138].time.Day := 13, [1138].time.Hour := 15, [1138].time.Minute := 14, [1138].time.Second := 59, [1139].log_data[0].min := 1.0, [1139].log_data[0].max := 1.0, [1139].log_data[0].total := 300.0, [1139].log_data[0].time := 300.0, [1139].log_data[0].minminute := 15, [1139].log_data[0].maxminute := 15, [1139].log_data[0].valid := 1, [1139].log_data[1].valid := 1, [1139].log_data[2].valid := 1, [1139].log_data[3].valid := 1, [1139].log_data[4].valid := 1, [1139].log_data[5].valid := 1, [1139].log_data[6].valid := 1, [1139].log_data[7].valid := 1, [1139].log_data[8].valid := 1, [1139].log_data[9].valid := 1, [1139].log_data[10].valid := 1, [1139].log_data[11].valid := 1, [1139].log_data[12].valid := 1, [1139].log_data[13].valid := 1, [1139].log_data[14].valid := 1, [1139].log_data[15].valid := 1, [1139].log_data[16].valid := 1, [1139].log_data[17].valid := 1, [1139].log_data[18].valid := 1, [1139].log_data[19].valid := 1, [1139].time.Year := 2023, [1139].time.Month := 1, [1139].time.Day := 13, [1139].time.Hour := 15, [1139].time.Minute := 19, [1139].time.Second := 59,
        [1140].log_data[0].min := 1.0, [1140].log_data[0].max := 1.0, [1140].log_data[0].total := 300.0, [1140].log_data[0].time := 300.0, [1140].log_data[0].minminute := 20, [1140].log_data[0].maxminute := 20, [1140].log_data[0].valid := 1, [1140].log_data[1].valid := 1, [1140].log_data[2].valid := 1, [1140].log_data[3].valid := 1, [1140].log_data[4].valid := 1, [1140].log_data[5].valid := 1, [1140].log_data[6].valid := 1, [1140].log_data[7].valid := 1, [1140].log_data[8].valid := 1, [1140].log_data[9].valid := 1, [1140].log_data[10].valid := 1, [1140].log_data[11].valid := 1, [1140].log_data[12].valid := 1, [1140].log_data[13].valid := 1, [1140].log_data[14].valid := 1, [1140].log_data[15].valid := 1, [1140].log_data[16].valid := 1, [1140].log_data[17].valid := 1, [1140].log_data[18].valid := 1, [1140].log_data[19].valid := 1, [1140].time.Year := 2023, [1140].time.Month := 1, [1140].time.Day := 13, [1140].time.Hour := 15, [1140].time.Minute := 24, [1140].time.Second := 59, [1141].log_data[0].min := 1.0, [1141].log_data[0].max := 1.0, [1141].log_data[0].total := 300.0, [1141].log_data[0].time := 300.0, [1141].log_data[0].minminute := 25, [1141].log_data[0].maxminute := 25, [1141].log_data[0].valid := 1, [1141].log_data[1].valid := 1, [1141].log_data[2].valid := 1, [1141].log_data[3].valid := 1, [1141].log_data[4].valid := 1, [1141].log_data[5].valid := 1, [1141].log_data[6].valid := 1, [1141].log_data[7].valid := 1, [1141].log_data[8].valid := 1, [1141].log_data[9].valid := 1, [1141].log_data[10].valid := 1, [1141].log_data[11].valid := 1, [1141].log_data[12].valid := 1, [1141].log_data[13].valid := 1, [1141].log_data[14].valid := 1, [1141].log_data[15].valid := 1, [1141].log_data[16].valid := 1, [1141].log_data[17].valid := 1, [1141].log_data[18].valid := 1, [1141].log_data[19].valid := 1, [1141].time.Year := 2023, [1141].time.Month := 1,
        [1141].time.Day := 13, [1141].time.Hour := 15, [1141].time.Minute := 29, [1141].time.Second := 59, [1142].log_data[0].min := 1.0, [1142].log_data[0].max := 1.0, [1142].log_data[0].total := 300.0, [1142].log_data[0].time := 300.0, [1142].log_data[0].minminute := 30, [1142].log_data[0].maxminute := 30, [1142].log_data[0].valid := 1, [1142].log_data[1].valid := 1, [1142].log_data[2].valid := 1, [1142].log_data[3].valid := 1, [1142].log_data[4].valid := 1, [1142].log_data[5].valid := 1, [1142].log_data[6].valid := 1, [1142].log_data[7].valid := 1, [1142].log_data[8].valid := 1, [1142].log_data[9].valid := 1, [1142].log_data[10].valid := 1, [1142].log_data[11].valid := 1, [1142].log_data[12].valid := 1, [1142].log_data[13].valid := 1, [1142].log_data[14].valid := 1, [1142].log_data[15].valid := 1, [1142].log_data[16].valid := 1, [1142].log_data[17].valid := 1, [1142].log_data[18].valid := 1, [1142].log_data[19].valid := 1, [1142].time.Year := 2023, [1142].time.Month := 1, [1142].time.Day := 13, [1142].time.Hour := 15, [1142].time.Minute := 34, [1142].time.Second := 59, [1143].log_data[0].min := 1.0, [1143].log_data[0].max := 1.0, [1143].log_data[0].total := 300.0, [1143].log_data[0].time := 300.0, [1143].log_data[0].minminute := 35, [1143].log_data[0].maxminute := 35, [1143].log_data[0].valid := 1, [1143].log_data[1].valid := 1, [1143].log_data[2].valid := 1, [1143].log_data[3].valid := 1, [1143].log_data[4].valid := 1, [1143].log_data[5].valid := 1, [1143].log_data[6].valid := 1, [1143].log_data[7].valid := 1, [1143].log_data[8].valid := 1, [1143].log_data[9].valid := 1, [1143].log_data[10].valid := 1, [1143].log_data[11].valid := 1, [1143].log_data[12].valid := 1, [1143].log_data[13].valid := 1, [1143].log_data[14].valid := 1, [1143].log_data[15].valid := 1, [1143].log_data[16].valid := 1, [1143].log_data[17].valid := 1,
        [1143].log_data[18].valid := 1, [1143].log_data[19].valid := 1, [1143].time.Year := 2023, [1143].time.Month := 1, [1143].time.Day := 13, [1143].time.Hour := 15, [1143].time.Minute := 39, [1143].time.Second := 59, [1144].log_data[0].min := 1.0, [1144].log_data[0].max := 1.0, [1144].log_data[0].total := 300.0, [1144].log_data[0].time := 300.0, [1144].log_data[0].minminute := 40, [1144].log_data[0].maxminute := 40, [1144].log_data[0].valid := 1, [1144].log_data[1].valid := 1, [1144].log_data[2].valid := 1, [1144].log_data[3].valid := 1, [1144].log_data[4].valid := 1, [1144].log_data[5].valid := 1, [1144].log_data[6].valid := 1, [1144].log_data[7].valid := 1, [1144].log_data[8].valid := 1, [1144].log_data[9].valid := 1, [1144].log_data[10].valid := 1, [1144].log_data[11].valid := 1, [1144].log_data[12].valid := 1, [1144].log_data[13].valid := 1, [1144].log_data[14].valid := 1, [1144].log_data[15].valid := 1, [1144].log_data[16].valid := 1, [1144].log_data[17].valid := 1, [1144].log_data[18].valid := 1, [1144].log_data[19].valid := 1, [1144].time.Year := 2023, [1144].time.Month := 1, [1144].time.Day := 13, [1144].time.Hour := 15, [1144].time.Minute := 44, [1144].time.Second := 59, [1145].log_data[0].min := 1.0, [1145].log_data[0].max := 1.0, [1145].log_data[0].total := 300.0, [1145].log_data[0].time := 300.0, [1145].log_data[0].minminute := 45, [1145].log_data[0].maxminute := 45, [1145].log_data[0].valid := 1, [1145].log_data[1].valid := 1, [1145].log_data[2].valid := 1, [1145].log_data[3].valid := 1, [1145].log_data[4].valid := 1, [1145].log_data[5].valid := 1, [1145].log_data[6].valid := 1, [1145].log_data[7].valid := 1, [1145].log_data[8].valid := 1, [1145].log_data[9].valid := 1, [1145].log_data[10].valid := 1, [1145].log_data[11].valid := 1, [1145].log_data[12].valid := 1, [1145].log_data[13].valid := 1,
        [1145].log_data[14].valid := 1, [1145].log_data[15].valid := 1, [1145].log_data[16].valid := 1, [1145].log_data[17].valid := 1, [1145].log_data[18].valid := 1, [1145].log_data[19].valid := 1, [1145].time.Year := 2023, [1145].time.Month := 1, [1145].time.Day := 13, [1145].time.Hour := 15, [1145].time.Minute := 49, [1145].time.Second := 59, [1146].log_data[0].min := 1.0, [1146].log_data[0].max := 1.0, [1146].log_data[0].total := 300.0, [1146].log_data[0].time := 300.0, [1146].log_data[0].minminute := 50, [1146].log_data[0].maxminute := 50, [1146].log_data[0].valid := 1, [1146].log_data[1].valid := 1, [1146].log_data[2].valid := 1, [1146].log_data[3].valid := 1, [1146].log_data[4].valid := 1, [1146].log_data[5].valid := 1, [1146].log_data[6].valid := 1, [1146].log_data[7].valid := 1, [1146].log_data[8].valid := 1, [1146].log_data[9].valid := 1, [1146].log_data[10].valid := 1, [1146].log_data[11].valid := 1, [1146].log_data[12].valid := 1, [1146].log_data[13].valid := 1, [1146].log_data[14].valid := 1, [1146].log_data[15].valid := 1, [1146].log_data[16].valid := 1, [1146].log_data[17].valid := 1, [1146].log_data[18].valid := 1, [1146].log_data[19].valid := 1, [1146].time.Year := 2023, [1146].time.Month := 1, [1146].time.Day := 13, [1146].time.Hour := 15, [1146].time.Minute := 54, [1146].time.Second := 59, [1147].log_data[0].min := 1.0, [1147].log_data[0].max := 1.0, [1147].log_data[0].total := 300.0, [1147].log_data[0].time := 300.0, [1147].log_data[0].minminute := 55, [1147].log_data[0].maxminute := 55, [1147].log_data[0].valid := 1, [1147].log_data[1].valid := 1, [1147].log_data[2].valid := 1, [1147].log_data[3].valid := 1, [1147].log_data[4].valid := 1, [1147].log_data[5].valid := 1, [1147].log_data[6].valid := 1, [1147].log_data[7].valid := 1, [1147].log_data[8].valid := 1, [1147].log_data[9].valid := 1,
        [1147].log_data[10].valid := 1, [1147].log_data[11].valid := 1, [1147].log_data[12].valid := 1, [1147].log_data[13].valid := 1, [1147].log_data[14].valid := 1, [1147].log_data[15].valid := 1, [1147].log_data[16].valid := 1, [1147].log_data[17].valid := 1, [1147].log_data[18].valid := 1, [1147].log_data[19].valid := 1, [1147].time.Year := 2023, [1147].time.Month := 1, [1147].time.Day := 13, [1147].time.Hour := 15, [1147].time.Minute := 59, [1147].time.Second := 59, [1148].log_data[0].min := 1.0, [1148].log_data[0].max := 1.0, [1148].log_data[0].total := 300.0, [1148].log_data[0].time := 300.0, [1148].log_data[0].valid := 1, [1148].log_data[1].valid := 1, [1148].log_data[2].valid := 1, [1148].log_data[3].valid := 1, [1148].log_data[4].valid := 1, [1148].log_data[5].valid := 1, [1148].log_data[6].valid := 1, [1148].log_data[7].valid := 1, [1148].log_data[8].valid := 1, [1148].log_data[9].valid := 1, [1148].log_data[10].valid := 1, [1148].log_data[11].valid := 1, [1148].log_data[12].valid := 1, [1148].log_data[13].valid := 1, [1148].log_data[14].valid := 1, [1148].log_data[15].valid := 1, [1148].log_data[16].valid := 1, [1148].log_data[17].valid := 1, [1148].log_data[18].valid := 1, [1148].log_data[19].valid := 1, [1148].time.Year := 2023, [1148].time.Month := 1, [1148].time.Day := 13, [1148].time.Hour := 16, [1148].time.Minute := 4, [1148].time.Second := 59, [1149].log_data[0].min := 1.0, [1149].log_data[0].max := 1.0, [1149].log_data[0].total := 300.0, [1149].log_data[0].time := 300.0, [1149].log_data[0].minminute := 5, [1149].log_data[0].maxminute := 5, [1149].log_data[0].valid := 1, [1149].log_data[1].valid := 1, [1149].log_data[2].valid := 1, [1149].log_data[3].valid := 1, [1149].log_data[4].valid := 1, [1149].log_data[5].valid := 1, [1149].log_data[6].valid := 1, [1149].log_data[7].valid := 1,
        [1149].log_data[8].valid := 1, [1149].log_data[9].valid := 1, [1149].log_data[10].valid := 1, [1149].log_data[11].valid := 1, [1149].log_data[12].valid := 1, [1149].log_data[13].valid := 1, [1149].log_data[14].valid := 1, [1149].log_data[15].valid := 1, [1149].log_data[16].valid := 1, [1149].log_data[17].valid := 1, [1149].log_data[18].valid := 1, [1149].log_data[19].valid := 1, [1149].time.Year := 2023, [1149].time.Month := 1, [1149].time.Day := 13, [1149].time.Hour := 16, [1149].time.Minute := 9, [1149].time.Second := 59, [1150].log_data[0].min := 1.0, [1150].log_data[0].max := 1.0, [1150].log_data[0].total := 300.0, [1150].log_data[0].time := 300.0, [1150].log_data[0].minminute := 10, [1150].log_data[0].maxminute := 10, [1150].log_data[0].valid := 1, [1150].log_data[1].valid := 1, [1150].log_data[2].valid := 1, [1150].log_data[3].valid := 1, [1150].log_data[4].valid := 1, [1150].log_data[5].valid := 1, [1150].log_data[6].valid := 1, [1150].log_data[7].valid := 1, [1150].log_data[8].valid := 1, [1150].log_data[9].valid := 1, [1150].log_data[10].valid := 1, [1150].log_data[11].valid := 1, [1150].log_data[12].valid := 1, [1150].log_data[13].valid := 1, [1150].log_data[14].valid := 1, [1150].log_data[15].valid := 1, [1150].log_data[16].valid := 1, [1150].log_data[17].valid := 1, [1150].log_data[18].valid := 1, [1150].log_data[19].valid := 1, [1150].time.Year := 2023, [1150].time.Month := 1, [1150].time.Day := 13, [1150].time.Hour := 16, [1150].time.Minute := 14, [1150].time.Second := 59, [1151].log_data[0].min := 1.0, [1151].log_data[0].max := 1.0, [1151].log_data[0].total := 300.0, [1151].log_data[0].time := 300.0, [1151].log_data[0].minminute := 15, [1151].log_data[0].maxminute := 15, [1151].log_data[0].valid := 1, [1151].log_data[1].valid := 1, [1151].log_data[2].valid := 1, [1151].log_data[3].valid := 1,
        [1151].log_data[4].valid := 1, [1151].log_data[5].valid := 1, [1151].log_data[6].valid := 1, [1151].log_data[7].valid := 1, [1151].log_data[8].valid := 1, [1151].log_data[9].valid := 1, [1151].log_data[10].valid := 1, [1151].log_data[11].valid := 1, [1151].log_data[12].valid := 1, [1151].log_data[13].valid := 1, [1151].log_data[14].valid := 1, [1151].log_data[15].valid := 1, [1151].log_data[16].valid := 1, [1151].log_data[17].valid := 1, [1151].log_data[18].valid := 1, [1151].log_data[19].valid := 1, [1151].time.Year := 2023, [1151].time.Month := 1, [1151].time.Day := 13, [1151].time.Hour := 16, [1151].time.Minute := 19, [1151].time.Second := 59, [1152].log_data[0].min := 1.0, [1152].log_data[0].max := 1.0, [1152].log_data[0].total := 300.0, [1152].log_data[0].time := 300.0, [1152].log_data[0].minminute := 20, [1152].log_data[0].maxminute := 20, [1152].log_data[0].valid := 1, [1152].log_data[1].valid := 1, [1152].log_data[2].valid := 1, [1152].log_data[3].valid := 1, [1152].log_data[4].valid := 1, [1152].log_data[5].valid := 1, [1152].log_data[6].valid := 1, [1152].log_data[7].valid := 1, [1152].log_data[8].valid := 1, [1152].log_data[9].valid := 1, [1152].log_data[10].valid := 1, [1152].log_data[11].valid := 1, [1152].log_data[12].valid := 1, [1152].log_data[13].valid := 1, [1152].log_data[14].valid := 1, [1152].log_data[15].valid := 1, [1152].log_data[16].valid := 1, [1152].log_data[17].valid := 1, [1152].log_data[18].valid := 1, [1152].log_data[19].valid := 1, [1152].time.Year := 2023, [1152].time.Month := 1, [1152].time.Day := 13, [1152].time.Hour := 16, [1152].time.Minute := 24, [1152].time.Second := 59, [1153].log_data[0].min := 1.0, [1153].log_data[0].max := 1.0, [1153].log_data[0].total := 300.0, [1153].log_data[0].time := 300.0, [1153].log_data[0].minminute := 25, [1153].log_data[0].maxminute := 25,
        [1153].log_data[0].valid := 1, [1153].log_data[1].valid := 1, [1153].log_data[2].valid := 1, [1153].log_data[3].valid := 1, [1153].log_data[4].valid := 1, [1153].log_data[5].valid := 1, [1153].log_data[6].valid := 1, [1153].log_data[7].valid := 1, [1153].log_data[8].valid := 1, [1153].log_data[9].valid := 1, [1153].log_data[10].valid := 1, [1153].log_data[11].valid := 1, [1153].log_data[12].valid := 1, [1153].log_data[13].valid := 1, [1153].log_data[14].valid := 1, [1153].log_data[15].valid := 1, [1153].log_data[16].valid := 1, [1153].log_data[17].valid := 1, [1153].log_data[18].valid := 1, [1153].log_data[19].valid := 1, [1153].time.Year := 2023, [1153].time.Month := 1, [1153].time.Day := 13, [1153].time.Hour := 16, [1153].time.Minute := 29, [1153].time.Second := 59, [1154].log_data[0].min := 1.0, [1154].log_data[0].max := 1.0, [1154].log_data[0].total := 300.0, [1154].log_data[0].time := 300.0, [1154].log_data[0].minminute := 30, [1154].log_data[0].maxminute := 30, [1154].log_data[0].valid := 1, [1154].log_data[1].valid := 1, [1154].log_data[2].valid := 1, [1154].log_data[3].valid := 1, [1154].log_data[4].valid := 1, [1154].log_data[5].valid := 1, [1154].log_data[6].valid := 1, [1154].log_data[7].valid := 1, [1154].log_data[8].valid := 1, [1154].log_data[9].valid := 1, [1154].log_data[10].valid := 1, [1154].log_data[11].valid := 1, [1154].log_data[12].valid := 1, [1154].log_data[13].valid := 1, [1154].log_data[14].valid := 1, [1154].log_data[15].valid := 1, [1154].log_data[16].valid := 1, [1154].log_data[17].valid := 1, [1154].log_data[18].valid := 1, [1154].log_data[19].valid := 1, [1154].time.Year := 2023, [1154].time.Month := 1, [1154].time.Day := 13, [1154].time.Hour := 16, [1154].time.Minute := 34, [1154].time.Second := 59, [1155].log_data[0].min := 1.0, [1155].log_data[0].max := 1.0,
        [1155].log_data[0].total := 300.0, [1155].log_data[0].time := 300.0, [1155].log_data[0].minminute := 35, [1155].log_data[0].maxminute := 35, [1155].log_data[0].valid := 1, [1155].log_data[1].valid := 1, [1155].log_data[2].valid := 1, [1155].log_data[3].valid := 1, [1155].log_data[4].valid := 1, [1155].log_data[5].valid := 1, [1155].log_data[6].valid := 1, [1155].log_data[7].valid := 1, [1155].log_data[8].valid := 1, [1155].log_data[9].valid := 1, [1155].log_data[10].valid := 1, [1155].log_data[11].valid := 1, [1155].log_data[12].valid := 1, [1155].log_data[13].valid := 1, [1155].log_data[14].valid := 1, [1155].log_data[15].valid := 1, [1155].log_data[16].valid := 1, [1155].log_data[17].valid := 1, [1155].log_data[18].valid := 1, [1155].log_data[19].valid := 1, [1155].time.Year := 2023, [1155].time.Month := 1, [1155].time.Day := 13, [1155].time.Hour := 16, [1155].time.Minute := 39, [1155].time.Second := 59, [1156].log_data[0].min := 1.0, [1156].log_data[0].max := 1.0, [1156].log_data[0].total := 300.0, [1156].log_data[0].time := 300.0, [1156].log_data[0].minminute := 40, [1156].log_data[0].maxminute := 40, [1156].log_data[0].valid := 1, [1156].log_data[1].valid := 1, [1156].log_data[2].valid := 1, [1156].log_data[3].valid := 1, [1156].log_data[4].valid := 1, [1156].log_data[5].valid := 1, [1156].log_data[6].valid := 1, [1156].log_data[7].valid := 1, [1156].log_data[8].valid := 1, [1156].log_data[9].valid := 1, [1156].log_data[10].valid := 1, [1156].log_data[11].valid := 1, [1156].log_data[12].valid := 1, [1156].log_data[13].valid := 1, [1156].log_data[14].valid := 1, [1156].log_data[15].valid := 1, [1156].log_data[16].valid := 1, [1156].log_data[17].valid := 1, [1156].log_data[18].valid := 1, [1156].log_data[19].valid := 1, [1156].time.Year := 2023, [1156].time.Month := 1, [1156].time.Day := 13, [1156].time.Hour := 16,
        [1156].time.Minute := 44, [1156].time.Second := 59, [1157].log_data[0].min := 1.0, [1157].log_data[0].max := 1.0, [1157].log_data[0].total := 300.0, [1157].log_data[0].time := 300.0, [1157].log_data[0].minminute := 45, [1157].log_data[0].maxminute := 45, [1157].log_data[0].valid := 1, [1157].log_data[1].valid := 1, [1157].log_data[2].valid := 1, [1157].log_data[3].valid := 1, [1157].log_data[4].valid := 1, [1157].log_data[5].valid := 1, [1157].log_data[6].valid := 1, [1157].log_data[7].valid := 1, [1157].log_data[8].valid := 1, [1157].log_data[9].valid := 1, [1157].log_data[10].valid := 1, [1157].log_data[11].valid := 1, [1157].log_data[12].valid := 1, [1157].log_data[13].valid := 1, [1157].log_data[14].valid := 1, [1157].log_data[15].valid := 1, [1157].log_data[16].valid := 1, [1157].log_data[17].valid := 1, [1157].log_data[18].valid := 1, [1157].log_data[19].valid := 1, [1157].time.Year := 2023, [1157].time.Month := 1, [1157].time.Day := 13, [1157].time.Hour := 16, [1157].time.Minute := 49, [1157].time.Second := 59, [1158].log_data[0].min := 1.0, [1158].log_data[0].max := 1.0, [1158].log_data[0].total := 300.0, [1158].log_data[0].time := 300.0, [1158].log_data[0].minminute := 50, [1158].log_data[0].maxminute := 50, [1158].log_data[0].valid := 1, [1158].log_data[1].valid := 1, [1158].log_data[2].valid := 1, [1158].log_data[3].valid := 1, [1158].log_data[4].valid := 1, [1158].log_data[5].valid := 1, [1158].log_data[6].valid := 1, [1158].log_data[7].valid := 1, [1158].log_data[8].valid := 1, [1158].log_data[9].valid := 1, [1158].log_data[10].valid := 1, [1158].log_data[11].valid := 1, [1158].log_data[12].valid := 1, [1158].log_data[13].valid := 1, [1158].log_data[14].valid := 1, [1158].log_data[15].valid := 1, [1158].log_data[16].valid := 1, [1158].log_data[17].valid := 1, [1158].log_data[18].valid := 1, [1158].log_data[19].valid := 1,
        [1158].time.Year := 2023, [1158].time.Month := 1, [1158].time.Day := 13, [1158].time.Hour := 16, [1158].time.Minute := 54, [1158].time.Second := 59, [1159].log_data[0].min := 1.0, [1159].log_data[0].max := 1.0, [1159].log_data[0].total := 300.0, [1159].log_data[0].time := 300.0, [1159].log_data[0].minminute := 55, [1159].log_data[0].maxminute := 55, [1159].log_data[0].valid := 1, [1159].log_data[1].valid := 1, [1159].log_data[2].valid := 1, [1159].log_data[3].valid := 1, [1159].log_data[4].valid := 1, [1159].log_data[5].valid := 1, [1159].log_data[6].valid := 1, [1159].log_data[7].valid := 1, [1159].log_data[8].valid := 1, [1159].log_data[9].valid := 1, [1159].log_data[10].valid := 1, [1159].log_data[11].valid := 1, [1159].log_data[12].valid := 1, [1159].log_data[13].valid := 1, [1159].log_data[14].valid := 1, [1159].log_data[15].valid := 1, [1159].log_data[16].valid := 1, [1159].log_data[17].valid := 1, [1159].log_data[18].valid := 1, [1159].log_data[19].valid := 1, [1159].time.Year := 2023, [1159].time.Month := 1, [1159].time.Day := 13, [1159].time.Hour := 16, [1159].time.Minute := 59, [1159].time.Second := 59, [1160].log_data[0].min := 1.0, [1160].log_data[0].max := 1.0, [1160].log_data[0].total := 300.0, [1160].log_data[0].time := 300.0, [1160].log_data[0].valid := 1, [1160].log_data[1].valid := 1, [1160].log_data[2].valid := 1, [1160].log_data[3].valid := 1, [1160].log_data[4].valid := 1, [1160].log_data[5].valid := 1, [1160].log_data[6].valid := 1, [1160].log_data[7].valid := 1, [1160].log_data[8].valid := 1, [1160].log_data[9].valid := 1, [1160].log_data[10].valid := 1, [1160].log_data[11].valid := 1, [1160].log_data[12].valid := 1, [1160].log_data[13].valid := 1, [1160].log_data[14].valid := 1, [1160].log_data[15].valid := 1, [1160].log_data[16].valid := 1, [1160].log_data[17].valid := 1,
        [1160].log_data[18].valid := 1, [1160].log_data[19].valid := 1, [1160].time.Year := 2023, [1160].time.Month := 1, [1160].time.Day := 13, [1160].time.Hour := 17, [1160].time.Minute := 4, [1160].time.Second := 59, [1161].log_data[0].min := 1.0, [1161].log_data[0].max := 1.0, [1161].log_data[0].total := 300.0, [1161].log_data[0].time := 300.0, [1161].log_data[0].minminute := 5, [1161].log_data[0].maxminute := 5, [1161].log_data[0].valid := 1, [1161].log_data[1].valid := 1, [1161].log_data[2].valid := 1, [1161].log_data[3].valid := 1, [1161].log_data[4].valid := 1, [1161].log_data[5].valid := 1, [1161].log_data[6].valid := 1, [1161].log_data[7].valid := 1, [1161].log_data[8].valid := 1, [1161].log_data[9].valid := 1, [1161].log_data[10].valid := 1, [1161].log_data[11].valid := 1, [1161].log_data[12].valid := 1, [1161].log_data[13].valid := 1, [1161].log_data[14].valid := 1, [1161].log_data[15].valid := 1, [1161].log_data[16].valid := 1, [1161].log_data[17].valid := 1, [1161].log_data[18].valid := 1, [1161].log_data[19].valid := 1, [1161].time.Year := 2023, [1161].time.Month := 1, [1161].time.Day := 13, [1161].time.Hour := 17, [1161].time.Minute := 9, [1161].time.Second := 59, [1162].log_data[0].min := 1.0, [1162].log_data[0].max := 1.0, [1162].log_data[0].total := 300.0, [1162].log_data[0].time := 300.0, [1162].log_data[0].minminute := 10, [1162].log_data[0].maxminute := 10, [1162].log_data[0].valid := 1, [1162].log_data[1].valid := 1, [1162].log_data[2].valid := 1, [1162].log_data[3].valid := 1, [1162].log_data[4].valid := 1, [1162].log_data[5].valid := 1, [1162].log_data[6].valid := 1, [1162].log_data[7].valid := 1, [1162].log_data[8].valid := 1, [1162].log_data[9].valid := 1, [1162].log_data[10].valid := 1, [1162].log_data[11].valid := 1, [1162].log_data[12].valid := 1, [1162].log_data[13].valid := 1,
        [1162].log_data[14].valid := 1, [1162].log_data[15].valid := 1, [1162].log_data[16].valid := 1, [1162].log_data[17].valid := 1, [1162].log_data[18].valid := 1, [1162].log_data[19].valid := 1, [1162].time.Year := 2023, [1162].time.Month := 1, [1162].time.Day := 13, [1162].time.Hour := 17, [1162].time.Minute := 14, [1162].time.Second := 59, [1163].log_data[0].min := 1.0, [1163].log_data[0].max := 1.0, [1163].log_data[0].total := 300.0, [1163].log_data[0].time := 300.0, [1163].log_data[0].minminute := 15, [1163].log_data[0].maxminute := 15, [1163].log_data[0].valid := 1, [1163].log_data[1].valid := 1, [1163].log_data[2].valid := 1, [1163].log_data[3].valid := 1, [1163].log_data[4].valid := 1, [1163].log_data[5].valid := 1, [1163].log_data[6].valid := 1, [1163].log_data[7].valid := 1, [1163].log_data[8].valid := 1, [1163].log_data[9].valid := 1, [1163].log_data[10].valid := 1, [1163].log_data[11].valid := 1, [1163].log_data[12].valid := 1, [1163].log_data[13].valid := 1, [1163].log_data[14].valid := 1, [1163].log_data[15].valid := 1, [1163].log_data[16].valid := 1, [1163].log_data[17].valid := 1, [1163].log_data[18].valid := 1, [1163].log_data[19].valid := 1, [1163].time.Year := 2023, [1163].time.Month := 1, [1163].time.Day := 13, [1163].time.Hour := 17, [1163].time.Minute := 19, [1163].time.Second := 59, [1164].log_data[0].min := 1.0, [1164].log_data[0].max := 1.0, [1164].log_data[0].total := 300.0, [1164].log_data[0].time := 300.0, [1164].log_data[0].minminute := 20, [1164].log_data[0].maxminute := 20, [1164].log_data[0].valid := 1, [1164].log_data[1].valid := 1, [1164].log_data[2].valid := 1, [1164].log_data[3].valid := 1, [1164].log_data[4].valid := 1, [1164].log_data[5].valid := 1, [1164].log_data[6].valid := 1, [1164].log_data[7].valid := 1, [1164].log_data[8].valid := 1, [1164].log_data[9].valid := 1,
        [1164].log_data[10].valid := 1, [1164].log_data[11].valid := 1, [1164].log_data[12].valid := 1, [1164].log_data[13].valid := 1, [1164].log_data[14].valid := 1, [1164].log_data[15].valid := 1, [1164].log_data[16].valid := 1, [1164].log_data[17].valid := 1, [1164].log_data[18].valid := 1, [1164].log_data[19].valid := 1, [1164].time.Year := 2023, [1164].time.Month := 1, [1164].time.Day := 13, [1164].time.Hour := 17, [1164].time.Minute := 24, [1164].time.Second := 59, [1165].log_data[0].min := 1.0, [1165].log_data[0].max := 1.0, [1165].log_data[0].total := 300.0, [1165].log_data[0].time := 300.0, [1165].log_data[0].minminute := 25, [1165].log_data[0].maxminute := 25, [1165].log_data[0].valid := 1, [1165].log_data[1].valid := 1, [1165].log_data[2].valid := 1, [1165].log_data[3].valid := 1, [1165].log_data[4].valid := 1, [1165].log_data[5].valid := 1, [1165].log_data[6].valid := 1, [1165].log_data[7].valid := 1, [1165].log_data[8].valid := 1, [1165].log_data[9].valid := 1, [1165].log_data[10].valid := 1, [1165].log_data[11].valid := 1, [1165].log_data[12].valid := 1, [1165].log_data[13].valid := 1, [1165].log_data[14].valid := 1, [1165].log_data[15].valid := 1, [1165].log_data[16].valid := 1, [1165].log_data[17].valid := 1, [1165].log_data[18].valid := 1, [1165].log_data[19].valid := 1, [1165].time.Year := 2023, [1165].time.Month := 1, [1165].time.Day := 13, [1165].time.Hour := 17, [1165].time.Minute := 29, [1165].time.Second := 59, [1166].log_data[0].min := 1.0, [1166].log_data[0].max := 1.0, [1166].log_data[0].total := 300.0, [1166].log_data[0].time := 300.0, [1166].log_data[0].minminute := 30, [1166].log_data[0].maxminute := 30, [1166].log_data[0].valid := 1, [1166].log_data[1].valid := 1, [1166].log_data[2].valid := 1, [1166].log_data[3].valid := 1, [1166].log_data[4].valid := 1, [1166].log_data[5].valid := 1,
        [1166].log_data[6].valid := 1, [1166].log_data[7].valid := 1, [1166].log_data[8].valid := 1, [1166].log_data[9].valid := 1, [1166].log_data[10].valid := 1, [1166].log_data[11].valid := 1, [1166].log_data[12].valid := 1, [1166].log_data[13].valid := 1, [1166].log_data[14].valid := 1, [1166].log_data[15].valid := 1, [1166].log_data[16].valid := 1, [1166].log_data[17].valid := 1, [1166].log_data[18].valid := 1, [1166].log_data[19].valid := 1, [1166].time.Year := 2023, [1166].time.Month := 1, [1166].time.Day := 13, [1166].time.Hour := 17, [1166].time.Minute := 34, [1166].time.Second := 59, [1167].log_data[0].min := 1.0, [1167].log_data[0].max := 1.0, [1167].log_data[0].total := 300.0, [1167].log_data[0].time := 300.0, [1167].log_data[0].minminute := 35, [1167].log_data[0].maxminute := 35, [1167].log_data[0].valid := 1, [1167].log_data[1].valid := 1, [1167].log_data[2].valid := 1, [1167].log_data[3].valid := 1, [1167].log_data[4].valid := 1, [1167].log_data[5].valid := 1, [1167].log_data[6].valid := 1, [1167].log_data[7].valid := 1, [1167].log_data[8].valid := 1, [1167].log_data[9].valid := 1, [1167].log_data[10].valid := 1, [1167].log_data[11].valid := 1, [1167].log_data[12].valid := 1, [1167].log_data[13].valid := 1, [1167].log_data[14].valid := 1, [1167].log_data[15].valid := 1, [1167].log_data[16].valid := 1, [1167].log_data[17].valid := 1, [1167].log_data[18].valid := 1, [1167].log_data[19].valid := 1, [1167].time.Year := 2023, [1167].time.Month := 1, [1167].time.Day := 13, [1167].time.Hour := 17, [1167].time.Minute := 39, [1167].time.Second := 59, [1168].log_data[0].min := 1.0, [1168].log_data[0].max := 1.0, [1168].log_data[0].total := 300.0, [1168].log_data[0].time := 300.0, [1168].log_data[0].minminute := 40, [1168].log_data[0].maxminute := 40, [1168].log_data[0].valid := 1, [1168].log_data[1].valid := 1,
        [1168].log_data[2].valid := 1, [1168].log_data[3].valid := 1, [1168].log_data[4].valid := 1, [1168].log_data[5].valid := 1, [1168].log_data[6].valid := 1, [1168].log_data[7].valid := 1, [1168].log_data[8].valid := 1, [1168].log_data[9].valid := 1, [1168].log_data[10].valid := 1, [1168].log_data[11].valid := 1, [1168].log_data[12].valid := 1, [1168].log_data[13].valid := 1, [1168].log_data[14].valid := 1, [1168].log_data[15].valid := 1, [1168].log_data[16].valid := 1, [1168].log_data[17].valid := 1, [1168].log_data[18].valid := 1, [1168].log_data[19].valid := 1, [1168].time.Year := 2023, [1168].time.Month := 1, [1168].time.Day := 13, [1168].time.Hour := 17, [1168].time.Minute := 44, [1168].time.Second := 59, [1169].log_data[0].min := 1.0, [1169].log_data[0].max := 1.0, [1169].log_data[0].total := 300.0, [1169].log_data[0].time := 300.0, [1169].log_data[0].minminute := 45, [1169].log_data[0].maxminute := 45, [1169].log_data[0].valid := 1, [1169].log_data[1].valid := 1, [1169].log_data[2].valid := 1, [1169].log_data[3].valid := 1, [1169].log_data[4].valid := 1, [1169].log_data[5].valid := 1, [1169].log_data[6].valid := 1, [1169].log_data[7].valid := 1, [1169].log_data[8].valid := 1, [1169].log_data[9].valid := 1, [1169].log_data[10].valid := 1, [1169].log_data[11].valid := 1, [1169].log_data[12].valid := 1, [1169].log_data[13].valid := 1, [1169].log_data[14].valid := 1, [1169].log_data[15].valid := 1, [1169].log_data[16].valid := 1, [1169].log_data[17].valid := 1, [1169].log_data[18].valid := 1, [1169].log_data[19].valid := 1, [1169].time.Year := 2023, [1169].time.Month := 1, [1169].time.Day := 13, [1169].time.Hour := 17, [1169].time.Minute := 49, [1169].time.Second := 59, [1170].log_data[0].min := 1.0, [1170].log_data[0].max := 1.0, [1170].log_data[0].total := 300.0, [1170].log_data[0].time := 300.0,
        [1170].log_data[0].minminute := 50, [1170].log_data[0].maxminute := 50, [1170].log_data[0].valid := 1, [1170].log_data[1].valid := 1, [1170].log_data[2].valid := 1, [1170].log_data[3].valid := 1, [1170].log_data[4].valid := 1, [1170].log_data[5].valid := 1, [1170].log_data[6].valid := 1, [1170].log_data[7].valid := 1, [1170].log_data[8].valid := 1, [1170].log_data[9].valid := 1, [1170].log_data[10].valid := 1, [1170].log_data[11].valid := 1, [1170].log_data[12].valid := 1, [1170].log_data[13].valid := 1, [1170].log_data[14].valid := 1, [1170].log_data[15].valid := 1, [1170].log_data[16].valid := 1, [1170].log_data[17].valid := 1, [1170].log_data[18].valid := 1, [1170].log_data[19].valid := 1, [1170].time.Year := 2023, [1170].time.Month := 1, [1170].time.Day := 13, [1170].time.Hour := 17, [1170].time.Minute := 54, [1170].time.Second := 59, [1171].log_data[0].min := 1.0, [1171].log_data[0].max := 1.0, [1171].log_data[0].total := 300.0, [1171].log_data[0].time := 300.0, [1171].log_data[0].minminute := 55, [1171].log_data[0].maxminute := 55, [1171].log_data[0].valid := 1, [1171].log_data[1].valid := 1, [1171].log_data[2].valid := 1, [1171].log_data[3].valid := 1, [1171].log_data[4].valid := 1, [1171].log_data[5].valid := 1, [1171].log_data[6].valid := 1, [1171].log_data[7].valid := 1, [1171].log_data[8].valid := 1, [1171].log_data[9].valid := 1, [1171].log_data[10].valid := 1, [1171].log_data[11].valid := 1, [1171].log_data[12].valid := 1, [1171].log_data[13].valid := 1, [1171].log_data[14].valid := 1, [1171].log_data[15].valid := 1, [1171].log_data[16].valid := 1, [1171].log_data[17].valid := 1, [1171].log_data[18].valid := 1, [1171].log_data[19].valid := 1, [1171].time.Year := 2023, [1171].time.Month := 1, [1171].time.Day := 13, [1171].time.Hour := 17, [1171].time.Minute := 59, [1171].time.Second := 59,
        [1172].log_data[0].min := 1.0, [1172].log_data[0].max := 1.0, [1172].log_data[0].total := 300.0, [1172].log_data[0].time := 300.0, [1172].log_data[0].valid := 1, [1172].log_data[1].valid := 1, [1172].log_data[2].valid := 1, [1172].log_data[3].valid := 1, [1172].log_data[4].valid := 1, [1172].log_data[5].valid := 1, [1172].log_data[6].valid := 1, [1172].log_data[7].valid := 1, [1172].log_data[8].valid := 1, [1172].log_data[9].valid := 1, [1172].log_data[10].valid := 1, [1172].log_data[11].valid := 1, [1172].log_data[12].valid := 1, [1172].log_data[13].valid := 1, [1172].log_data[14].valid := 1, [1172].log_data[15].valid := 1, [1172].log_data[16].valid := 1, [1172].log_data[17].valid := 1, [1172].log_data[18].valid := 1, [1172].log_data[19].valid := 1, [1172].time.Year := 2023, [1172].time.Month := 1, [1172].time.Day := 13, [1172].time.Hour := 18, [1172].time.Minute := 4, [1172].time.Second := 59, [1173].log_data[0].min := 1.0, [1173].log_data[0].max := 1.0, [1173].log_data[0].total := 300.0, [1173].log_data[0].time := 300.0, [1173].log_data[0].minminute := 5, [1173].log_data[0].maxminute := 5, [1173].log_data[0].valid := 1, [1173].log_data[1].valid := 1, [1173].log_data[2].valid := 1, [1173].log_data[3].valid := 1, [1173].log_data[4].valid := 1, [1173].log_data[5].valid := 1, [1173].log_data[6].valid := 1, [1173].log_data[7].valid := 1, [1173].log_data[8].valid := 1, [1173].log_data[9].valid := 1, [1173].log_data[10].valid := 1, [1173].log_data[11].valid := 1, [1173].log_data[12].valid := 1, [1173].log_data[13].valid := 1, [1173].log_data[14].valid := 1, [1173].log_data[15].valid := 1, [1173].log_data[16].valid := 1, [1173].log_data[17].valid := 1, [1173].log_data[18].valid := 1, [1173].log_data[19].valid := 1, [1173].time.Year := 2023, [1173].time.Month := 1, [1173].time.Day := 13, [1173].time.Hour := 18,
        [1173].time.Minute := 9, [1173].time.Second := 59, [1174].log_data[0].min := 1.0, [1174].log_data[0].max := 1.0, [1174].log_data[0].total := 300.0, [1174].log_data[0].time := 300.0, [1174].log_data[0].minminute := 10, [1174].log_data[0].maxminute := 10, [1174].log_data[0].valid := 1, [1174].log_data[1].valid := 1, [1174].log_data[2].valid := 1, [1174].log_data[3].valid := 1, [1174].log_data[4].valid := 1, [1174].log_data[5].valid := 1, [1174].log_data[6].valid := 1, [1174].log_data[7].valid := 1, [1174].log_data[8].valid := 1, [1174].log_data[9].valid := 1, [1174].log_data[10].valid := 1, [1174].log_data[11].valid := 1, [1174].log_data[12].valid := 1, [1174].log_data[13].valid := 1, [1174].log_data[14].valid := 1, [1174].log_data[15].valid := 1, [1174].log_data[16].valid := 1, [1174].log_data[17].valid := 1, [1174].log_data[18].valid := 1, [1174].log_data[19].valid := 1, [1174].time.Year := 2023, [1174].time.Month := 1, [1174].time.Day := 13, [1174].time.Hour := 18, [1174].time.Minute := 14, [1174].time.Second := 59, [1175].log_data[0].min := 1.0, [1175].log_data[0].max := 1.0, [1175].log_data[0].total := 300.0, [1175].log_data[0].time := 300.0, [1175].log_data[0].minminute := 15, [1175].log_data[0].maxminute := 15, [1175].log_data[0].valid := 1, [1175].log_data[1].valid := 1, [1175].log_data[2].valid := 1, [1175].log_data[3].valid := 1, [1175].log_data[4].valid := 1, [1175].log_data[5].valid := 1, [1175].log_data[6].valid := 1, [1175].log_data[7].valid := 1, [1175].log_data[8].valid := 1, [1175].log_data[9].valid := 1, [1175].log_data[10].valid := 1, [1175].log_data[11].valid := 1, [1175].log_data[12].valid := 1, [1175].log_data[13].valid := 1, [1175].log_data[14].valid := 1, [1175].log_data[15].valid := 1, [1175].log_data[16].valid := 1, [1175].log_data[17].valid := 1, [1175].log_data[18].valid := 1, [1175].log_data[19].valid := 1,
        [1175].time.Year := 2023, [1175].time.Month := 1, [1175].time.Day := 13, [1175].time.Hour := 18, [1175].time.Minute := 19, [1175].time.Second := 59, [1176].log_data[0].min := 1.0, [1176].log_data[0].max := 1.0, [1176].log_data[0].total := 300.0, [1176].log_data[0].time := 300.0, [1176].log_data[0].minminute := 20, [1176].log_data[0].maxminute := 20, [1176].log_data[0].valid := 1, [1176].log_data[1].valid := 1, [1176].log_data[2].valid := 1, [1176].log_data[3].valid := 1, [1176].log_data[4].valid := 1, [1176].log_data[5].valid := 1, [1176].log_data[6].valid := 1, [1176].log_data[7].valid := 1, [1176].log_data[8].valid := 1, [1176].log_data[9].valid := 1, [1176].log_data[10].valid := 1, [1176].log_data[11].valid := 1, [1176].log_data[12].valid := 1, [1176].log_data[13].valid := 1, [1176].log_data[14].valid := 1, [1176].log_data[15].valid := 1, [1176].log_data[16].valid := 1, [1176].log_data[17].valid := 1, [1176].log_data[18].valid := 1, [1176].log_data[19].valid := 1, [1176].time.Year := 2023, [1176].time.Month := 1, [1176].time.Day := 13, [1176].time.Hour := 18, [1176].time.Minute := 24, [1176].time.Second := 59, [1177].log_data[0].min := 1.0, [1177].log_data[0].max := 1.0, [1177].log_data[0].total := 300.0, [1177].log_data[0].time := 300.0, [1177].log_data[0].minminute := 25, [1177].log_data[0].maxminute := 25, [1177].log_data[0].valid := 1, [1177].log_data[1].valid := 1, [1177].log_data[2].valid := 1, [1177].log_data[3].valid := 1, [1177].log_data[4].valid := 1, [1177].log_data[5].valid := 1, [1177].log_data[6].valid := 1, [1177].log_data[7].valid := 1, [1177].log_data[8].valid := 1, [1177].log_data[9].valid := 1, [1177].log_data[10].valid := 1, [1177].log_data[11].valid := 1, [1177].log_data[12].valid := 1, [1177].log_data[13].valid := 1, [1177].log_data[14].valid := 1, [1177].log_data[15].valid := 1,
        [1177].log_data[16].valid := 1, [1177].log_data[17].valid := 1, [1177].log_data[18].valid := 1, [1177].log_data[19].valid := 1, [1177].time.Year := 2023, [1177].time.Month := 1, [1177].time.Day := 13, [1177].time.Hour := 18, [1177].time.Minute := 29, [1177].time.Second := 59, [1178].log_data[0].min := 1.0, [1178].log_data[0].max := 1.0, [1178].log_data[0].total := 300.0, [1178].log_data[0].time := 300.0, [1178].log_data[0].minminute := 30, [1178].log_data[0].maxminute := 30, [1178].log_data[0].valid := 1, [1178].log_data[1].valid := 1, [1178].log_data[2].valid := 1, [1178].log_data[3].valid := 1, [1178].log_data[4].valid := 1, [1178].log_data[5].valid := 1, [1178].log_data[6].valid := 1, [1178].log_data[7].valid := 1, [1178].log_data[8].valid := 1, [1178].log_data[9].valid := 1, [1178].log_data[10].valid := 1, [1178].log_data[11].valid := 1, [1178].log_data[12].valid := 1, [1178].log_data[13].valid := 1, [1178].log_data[14].valid := 1, [1178].log_data[15].valid := 1, [1178].log_data[16].valid := 1, [1178].log_data[17].valid := 1, [1178].log_data[18].valid := 1, [1178].log_data[19].valid := 1, [1178].time.Year := 2023, [1178].time.Month := 1, [1178].time.Day := 13, [1178].time.Hour := 18, [1178].time.Minute := 34, [1178].time.Second := 59, [1179].log_data[0].min := 1.0, [1179].log_data[0].max := 1.0, [1179].log_data[0].total := 300.0, [1179].log_data[0].time := 300.0, [1179].log_data[0].minminute := 35, [1179].log_data[0].maxminute := 35, [1179].log_data[0].valid := 1, [1179].log_data[1].valid := 1, [1179].log_data[2].valid := 1, [1179].log_data[3].valid := 1, [1179].log_data[4].valid := 1, [1179].log_data[5].valid := 1, [1179].log_data[6].valid := 1, [1179].log_data[7].valid := 1, [1179].log_data[8].valid := 1, [1179].log_data[9].valid := 1, [1179].log_data[10].valid := 1, [1179].log_data[11].valid := 1,
        [1179].log_data[12].valid := 1, [1179].log_data[13].valid := 1, [1179].log_data[14].valid := 1, [1179].log_data[15].valid := 1, [1179].log_data[16].valid := 1, [1179].log_data[17].valid := 1, [1179].log_data[18].valid := 1, [1179].log_data[19].valid := 1, [1179].time.Year := 2023, [1179].time.Month := 1, [1179].time.Day := 13, [1179].time.Hour := 18, [1179].time.Minute := 39, [1179].time.Second := 59, [1180].log_data[0].min := 1.0, [1180].log_data[0].max := 1.0, [1180].log_data[0].total := 300.0, [1180].log_data[0].time := 300.0, [1180].log_data[0].minminute := 40, [1180].log_data[0].maxminute := 40, [1180].log_data[0].valid := 1, [1180].log_data[1].valid := 1, [1180].log_data[2].valid := 1, [1180].log_data[3].valid := 1, [1180].log_data[4].valid := 1, [1180].log_data[5].valid := 1, [1180].log_data[6].valid := 1, [1180].log_data[7].valid := 1, [1180].log_data[8].valid := 1, [1180].log_data[9].valid := 1, [1180].log_data[10].valid := 1, [1180].log_data[11].valid := 1, [1180].log_data[12].valid := 1, [1180].log_data[13].valid := 1, [1180].log_data[14].valid := 1, [1180].log_data[15].valid := 1, [1180].log_data[16].valid := 1, [1180].log_data[17].valid := 1, [1180].log_data[18].valid := 1, [1180].log_data[19].valid := 1, [1180].time.Year := 2023, [1180].time.Month := 1, [1180].time.Day := 13, [1180].time.Hour := 18, [1180].time.Minute := 44, [1180].time.Second := 59, [1181].log_data[0].min := 1.0, [1181].log_data[0].max := 1.0, [1181].log_data[0].total := 300.0, [1181].log_data[0].time := 300.0, [1181].log_data[0].minminute := 45, [1181].log_data[0].maxminute := 45, [1181].log_data[0].valid := 1, [1181].log_data[1].valid := 1, [1181].log_data[2].valid := 1, [1181].log_data[3].valid := 1, [1181].log_data[4].valid := 1, [1181].log_data[5].valid := 1, [1181].log_data[6].valid := 1, [1181].log_data[7].valid := 1,
        [1181].log_data[8].valid := 1, [1181].log_data[9].valid := 1, [1181].log_data[10].valid := 1, [1181].log_data[11].valid := 1, [1181].log_data[12].valid := 1, [1181].log_data[13].valid := 1, [1181].log_data[14].valid := 1, [1181].log_data[15].valid := 1, [1181].log_data[16].valid := 1, [1181].log_data[17].valid := 1, [1181].log_data[18].valid := 1, [1181].log_data[19].valid := 1, [1181].time.Year := 2023, [1181].time.Month := 1, [1181].time.Day := 13, [1181].time.Hour := 18, [1181].time.Minute := 49, [1181].time.Second := 59, [1182].log_data[0].min := 1.0, [1182].log_data[0].max := 1.0, [1182].log_data[0].total := 300.0, [1182].log_data[0].time := 300.0, [1182].log_data[0].minminute := 50, [1182].log_data[0].maxminute := 50, [1182].log_data[0].valid := 1, [1182].log_data[1].valid := 1, [1182].log_data[2].valid := 1, [1182].log_data[3].valid := 1, [1182].log_data[4].valid := 1, [1182].log_data[5].valid := 1, [1182].log_data[6].valid := 1, [1182].log_data[7].valid := 1, [1182].log_data[8].valid := 1, [1182].log_data[9].valid := 1, [1182].log_data[10].valid := 1, [1182].log_data[11].valid := 1, [1182].log_data[12].valid := 1, [1182].log_data[13].valid := 1, [1182].log_data[14].valid := 1, [1182].log_data[15].valid := 1, [1182].log_data[16].valid := 1, [1182].log_data[17].valid := 1, [1182].log_data[18].valid := 1, [1182].log_data[19].valid := 1, [1182].time.Year := 2023, [1182].time.Month := 1, [1182].time.Day := 13, [1182].time.Hour := 18, [1182].time.Minute := 54, [1182].time.Second := 59, [1183].log_data[0].min := 1.0, [1183].log_data[0].max := 1.0, [1183].log_data[0].total := 300.0, [1183].log_data[0].time := 300.0, [1183].log_data[0].minminute := 55, [1183].log_data[0].maxminute := 55, [1183].log_data[0].valid := 1, [1183].log_data[1].valid := 1, [1183].log_data[2].valid := 1, [1183].log_data[3].valid := 1,
        [1183].log_data[4].valid := 1, [1183].log_data[5].valid := 1, [1183].log_data[6].valid := 1, [1183].log_data[7].valid := 1, [1183].log_data[8].valid := 1, [1183].log_data[9].valid := 1, [1183].log_data[10].valid := 1, [1183].log_data[11].valid := 1, [1183].log_data[12].valid := 1, [1183].log_data[13].valid := 1, [1183].log_data[14].valid := 1, [1183].log_data[15].valid := 1, [1183].log_data[16].valid := 1, [1183].log_data[17].valid := 1, [1183].log_data[18].valid := 1, [1183].log_data[19].valid := 1, [1183].time.Year := 2023, [1183].time.Month := 1, [1183].time.Day := 13, [1183].time.Hour := 18, [1183].time.Minute := 59, [1183].time.Second := 59, [1184].log_data[0].min := 1.0, [1184].log_data[0].max := 1.0, [1184].log_data[0].total := 300.0, [1184].log_data[0].time := 300.0, [1184].log_data[0].valid := 1, [1184].log_data[1].valid := 1, [1184].log_data[2].valid := 1, [1184].log_data[3].valid := 1, [1184].log_data[4].valid := 1, [1184].log_data[5].valid := 1, [1184].log_data[6].valid := 1, [1184].log_data[7].valid := 1, [1184].log_data[8].valid := 1, [1184].log_data[9].valid := 1, [1184].log_data[10].valid := 1, [1184].log_data[11].valid := 1, [1184].log_data[12].valid := 1, [1184].log_data[13].valid := 1, [1184].log_data[14].valid := 1, [1184].log_data[15].valid := 1, [1184].log_data[16].valid := 1, [1184].log_data[17].valid := 1, [1184].log_data[18].valid := 1, [1184].log_data[19].valid := 1, [1184].time.Year := 2023, [1184].time.Month := 1, [1184].time.Day := 13, [1184].time.Hour := 19, [1184].time.Minute := 4, [1184].time.Second := 59, [1185].log_data[0].min := 1.0, [1185].log_data[0].max := 1.0, [1185].log_data[0].total := 300.0, [1185].log_data[0].time := 300.0, [1185].log_data[0].minminute := 5, [1185].log_data[0].maxminute := 5, [1185].log_data[0].valid := 1, [1185].log_data[1].valid := 1,
        [1185].log_data[2].valid := 1, [1185].log_data[3].valid := 1, [1185].log_data[4].valid := 1, [1185].log_data[5].valid := 1, [1185].log_data[6].valid := 1, [1185].log_data[7].valid := 1, [1185].log_data[8].valid := 1, [1185].log_data[9].valid := 1, [1185].log_data[10].valid := 1, [1185].log_data[11].valid := 1, [1185].log_data[12].valid := 1, [1185].log_data[13].valid := 1, [1185].log_data[14].valid := 1, [1185].log_data[15].valid := 1, [1185].log_data[16].valid := 1, [1185].log_data[17].valid := 1, [1185].log_data[18].valid := 1, [1185].log_data[19].valid := 1, [1185].time.Year := 2023, [1185].time.Month := 1, [1185].time.Day := 13, [1185].time.Hour := 19, [1185].time.Minute := 9, [1185].time.Second := 59, [1186].log_data[0].min := 1.0, [1186].log_data[0].max := 1.0, [1186].log_data[0].total := 300.0, [1186].log_data[0].time := 300.0, [1186].log_data[0].minminute := 10, [1186].log_data[0].maxminute := 10, [1186].log_data[0].valid := 1, [1186].log_data[1].valid := 1, [1186].log_data[2].valid := 1, [1186].log_data[3].valid := 1, [1186].log_data[4].valid := 1, [1186].log_data[5].valid := 1, [1186].log_data[6].valid := 1, [1186].log_data[7].valid := 1, [1186].log_data[8].valid := 1, [1186].log_data[9].valid := 1, [1186].log_data[10].valid := 1, [1186].log_data[11].valid := 1, [1186].log_data[12].valid := 1, [1186].log_data[13].valid := 1, [1186].log_data[14].valid := 1, [1186].log_data[15].valid := 1, [1186].log_data[16].valid := 1, [1186].log_data[17].valid := 1, [1186].log_data[18].valid := 1, [1186].log_data[19].valid := 1, [1186].time.Year := 2023, [1186].time.Month := 1, [1186].time.Day := 13, [1186].time.Hour := 19, [1186].time.Minute := 14, [1186].time.Second := 59, [1187].log_data[0].min := 1.0, [1187].log_data[0].max := 1.0, [1187].log_data[0].total := 300.0, [1187].log_data[0].time := 300.0,
        [1187].log_data[0].minminute := 15, [1187].log_data[0].maxminute := 15, [1187].log_data[0].valid := 1, [1187].log_data[1].valid := 1, [1187].log_data[2].valid := 1, [1187].log_data[3].valid := 1, [1187].log_data[4].valid := 1, [1187].log_data[5].valid := 1, [1187].log_data[6].valid := 1, [1187].log_data[7].valid := 1, [1187].log_data[8].valid := 1, [1187].log_data[9].valid := 1, [1187].log_data[10].valid := 1, [1187].log_data[11].valid := 1, [1187].log_data[12].valid := 1, [1187].log_data[13].valid := 1, [1187].log_data[14].valid := 1, [1187].log_data[15].valid := 1, [1187].log_data[16].valid := 1, [1187].log_data[17].valid := 1, [1187].log_data[18].valid := 1, [1187].log_data[19].valid := 1, [1187].time.Year := 2023, [1187].time.Month := 1, [1187].time.Day := 13, [1187].time.Hour := 19, [1187].time.Minute := 19, [1187].time.Second := 59, [1188].log_data[0].min := 1.0, [1188].log_data[0].max := 1.0, [1188].log_data[0].total := 300.0, [1188].log_data[0].time := 300.0, [1188].log_data[0].minminute := 20, [1188].log_data[0].maxminute := 20, [1188].log_data[0].valid := 1, [1188].log_data[1].valid := 1, [1188].log_data[2].valid := 1, [1188].log_data[3].valid := 1, [1188].log_data[4].valid := 1, [1188].log_data[5].valid := 1, [1188].log_data[6].valid := 1, [1188].log_data[7].valid := 1, [1188].log_data[8].valid := 1, [1188].log_data[9].valid := 1, [1188].log_data[10].valid := 1, [1188].log_data[11].valid := 1, [1188].log_data[12].valid := 1, [1188].log_data[13].valid := 1, [1188].log_data[14].valid := 1, [1188].log_data[15].valid := 1, [1188].log_data[16].valid := 1, [1188].log_data[17].valid := 1, [1188].log_data[18].valid := 1, [1188].log_data[19].valid := 1, [1188].time.Year := 2023, [1188].time.Month := 1, [1188].time.Day := 13, [1188].time.Hour := 19, [1188].time.Minute := 24, [1188].time.Second := 59,
        [1189].log_data[0].min := 1.0, [1189].log_data[0].max := 1.0, [1189].log_data[0].total := 300.0, [1189].log_data[0].time := 300.0, [1189].log_data[0].minminute := 25, [1189].log_data[0].maxminute := 25, [1189].log_data[0].valid := 1, [1189].log_data[1].valid := 1, [1189].log_data[2].valid := 1, [1189].log_data[3].valid := 1, [1189].log_data[4].valid := 1, [1189].log_data[5].valid := 1, [1189].log_data[6].valid := 1, [1189].log_data[7].valid := 1, [1189].log_data[8].valid := 1, [1189].log_data[9].valid := 1, [1189].log_data[10].valid := 1, [1189].log_data[11].valid := 1, [1189].log_data[12].valid := 1, [1189].log_data[13].valid := 1, [1189].log_data[14].valid := 1, [1189].log_data[15].valid := 1, [1189].log_data[16].valid := 1, [1189].log_data[17].valid := 1, [1189].log_data[18].valid := 1, [1189].log_data[19].valid := 1, [1189].time.Year := 2023, [1189].time.Month := 1, [1189].time.Day := 13, [1189].time.Hour := 19, [1189].time.Minute := 29, [1189].time.Second := 59, [1190].log_data[0].min := 1.0, [1190].log_data[0].max := 1.0, [1190].log_data[0].total := 300.0, [1190].log_data[0].time := 300.0, [1190].log_data[0].minminute := 30, [1190].log_data[0].maxminute := 30, [1190].log_data[0].valid := 1, [1190].log_data[1].valid := 1, [1190].log_data[2].valid := 1, [1190].log_data[3].valid := 1, [1190].log_data[4].valid := 1, [1190].log_data[5].valid := 1, [1190].log_data[6].valid := 1, [1190].log_data[7].valid := 1, [1190].log_data[8].valid := 1, [1190].log_data[9].valid := 1, [1190].log_data[10].valid := 1, [1190].log_data[11].valid := 1, [1190].log_data[12].valid := 1, [1190].log_data[13].valid := 1, [1190].log_data[14].valid := 1, [1190].log_data[15].valid := 1, [1190].log_data[16].valid := 1, [1190].log_data[17].valid := 1, [1190].log_data[18].valid := 1, [1190].log_data[19].valid := 1, [1190].time.Year := 2023, [1190].time.Month := 1,
        [1190].time.Day := 13, [1190].time.Hour := 19, [1190].time.Minute := 34, [1190].time.Second := 59, [1191].log_data[0].min := 1.0, [1191].log_data[0].max := 1.0, [1191].log_data[0].total := 300.0, [1191].log_data[0].time := 300.0, [1191].log_data[0].minminute := 35, [1191].log_data[0].maxminute := 35, [1191].log_data[0].valid := 1, [1191].log_data[1].valid := 1, [1191].log_data[2].valid := 1, [1191].log_data[3].valid := 1, [1191].log_data[4].valid := 1, [1191].log_data[5].valid := 1, [1191].log_data[6].valid := 1, [1191].log_data[7].valid := 1, [1191].log_data[8].valid := 1, [1191].log_data[9].valid := 1, [1191].log_data[10].valid := 1, [1191].log_data[11].valid := 1, [1191].log_data[12].valid := 1, [1191].log_data[13].valid := 1, [1191].log_data[14].valid := 1, [1191].log_data[15].valid := 1, [1191].log_data[16].valid := 1, [1191].log_data[17].valid := 1, [1191].log_data[18].valid := 1, [1191].log_data[19].valid := 1, [1191].time.Year := 2023, [1191].time.Month := 1, [1191].time.Day := 13, [1191].time.Hour := 19, [1191].time.Minute := 39, [1191].time.Second := 59, [1192].log_data[0].min := 1.0, [1192].log_data[0].max := 1.0, [1192].log_data[0].total := 300.0, [1192].log_data[0].time := 300.0, [1192].log_data[0].minminute := 40, [1192].log_data[0].maxminute := 40, [1192].log_data[0].valid := 1, [1192].log_data[1].valid := 1, [1192].log_data[2].valid := 1, [1192].log_data[3].valid := 1, [1192].log_data[4].valid := 1, [1192].log_data[5].valid := 1, [1192].log_data[6].valid := 1, [1192].log_data[7].valid := 1, [1192].log_data[8].valid := 1, [1192].log_data[9].valid := 1, [1192].log_data[10].valid := 1, [1192].log_data[11].valid := 1, [1192].log_data[12].valid := 1, [1192].log_data[13].valid := 1, [1192].log_data[14].valid := 1, [1192].log_data[15].valid := 1, [1192].log_data[16].valid := 1, [1192].log_data[17].valid := 1,
        [1192].log_data[18].valid := 1, [1192].log_data[19].valid := 1, [1192].time.Year := 2023, [1192].time.Month := 1, [1192].time.Day := 13, [1192].time.Hour := 19, [1192].time.Minute := 44, [1192].time.Second := 59, [1193].log_data[0].min := 1.0, [1193].log_data[0].max := 1.0, [1193].log_data[0].total := 300.0, [1193].log_data[0].time := 300.0, [1193].log_data[0].minminute := 45, [1193].log_data[0].maxminute := 45, [1193].log_data[0].valid := 1, [1193].log_data[1].valid := 1, [1193].log_data[2].valid := 1, [1193].log_data[3].valid := 1, [1193].log_data[4].valid := 1, [1193].log_data[5].valid := 1, [1193].log_data[6].valid := 1, [1193].log_data[7].valid := 1, [1193].log_data[8].valid := 1, [1193].log_data[9].valid := 1, [1193].log_data[10].valid := 1, [1193].log_data[11].valid := 1, [1193].log_data[12].valid := 1, [1193].log_data[13].valid := 1, [1193].log_data[14].valid := 1, [1193].log_data[15].valid := 1, [1193].log_data[16].valid := 1, [1193].log_data[17].valid := 1, [1193].log_data[18].valid := 1, [1193].log_data[19].valid := 1, [1193].time.Year := 2023, [1193].time.Month := 1, [1193].time.Day := 13, [1193].time.Hour := 19, [1193].time.Minute := 49, [1193].time.Second := 59, [1194].log_data[0].min := 1.0, [1194].log_data[0].max := 1.0, [1194].log_data[0].total := 300.0, [1194].log_data[0].time := 300.0, [1194].log_data[0].minminute := 50, [1194].log_data[0].maxminute := 50, [1194].log_data[0].valid := 1, [1194].log_data[1].valid := 1, [1194].log_data[2].valid := 1, [1194].log_data[3].valid := 1, [1194].log_data[4].valid := 1, [1194].log_data[5].valid := 1, [1194].log_data[6].valid := 1, [1194].log_data[7].valid := 1, [1194].log_data[8].valid := 1, [1194].log_data[9].valid := 1, [1194].log_data[10].valid := 1, [1194].log_data[11].valid := 1, [1194].log_data[12].valid := 1, [1194].log_data[13].valid := 1,
        [1194].log_data[14].valid := 1, [1194].log_data[15].valid := 1, [1194].log_data[16].valid := 1, [1194].log_data[17].valid := 1, [1194].log_data[18].valid := 1, [1194].log_data[19].valid := 1, [1194].time.Year := 2023, [1194].time.Month := 1, [1194].time.Day := 13, [1194].time.Hour := 19, [1194].time.Minute := 54, [1194].time.Second := 59, [1195].log_data[0].min := 1.0, [1195].log_data[0].max := 1.0, [1195].log_data[0].total := 300.0, [1195].log_data[0].time := 300.0, [1195].log_data[0].minminute := 55, [1195].log_data[0].maxminute := 55, [1195].log_data[0].valid := 1, [1195].log_data[1].valid := 1, [1195].log_data[2].valid := 1, [1195].log_data[3].valid := 1, [1195].log_data[4].valid := 1, [1195].log_data[5].valid := 1, [1195].log_data[6].valid := 1, [1195].log_data[7].valid := 1, [1195].log_data[8].valid := 1, [1195].log_data[9].valid := 1, [1195].log_data[10].valid := 1, [1195].log_data[11].valid := 1, [1195].log_data[12].valid := 1, [1195].log_data[13].valid := 1, [1195].log_data[14].valid := 1, [1195].log_data[15].valid := 1, [1195].log_data[16].valid := 1, [1195].log_data[17].valid := 1, [1195].log_data[18].valid := 1, [1195].log_data[19].valid := 1, [1195].time.Year := 2023, [1195].time.Month := 1, [1195].time.Day := 13, [1195].time.Hour := 19, [1195].time.Minute := 59, [1195].time.Second := 59, [1196].log_data[0].min := 1.0, [1196].log_data[0].max := 1.0, [1196].log_data[0].total := 300.0, [1196].log_data[0].time := 300.0, [1196].log_data[0].valid := 1, [1196].log_data[1].valid := 1, [1196].log_data[2].valid := 1, [1196].log_data[3].valid := 1, [1196].log_data[4].valid := 1, [1196].log_data[5].valid := 1, [1196].log_data[6].valid := 1, [1196].log_data[7].valid := 1, [1196].log_data[8].valid := 1, [1196].log_data[9].valid := 1, [1196].log_data[10].valid := 1, [1196].log_data[11].valid := 1,
        [1196].log_data[12].valid := 1, [1196].log_data[13].valid := 1, [1196].log_data[14].valid := 1, [1196].log_data[15].valid := 1, [1196].log_data[16].valid := 1, [1196].log_data[17].valid := 1, [1196].log_data[18].valid := 1, [1196].log_data[19].valid := 1, [1196].time.Year := 2023, [1196].time.Month := 1, [1196].time.Day := 13, [1196].time.Hour := 20, [1196].time.Minute := 4, [1196].time.Second := 59, [1197].log_data[0].min := 1.0, [1197].log_data[0].max := 1.0, [1197].log_data[0].total := 300.0, [1197].log_data[0].time := 300.0, [1197].log_data[0].minminute := 5, [1197].log_data[0].maxminute := 5, [1197].log_data[0].valid := 1, [1197].log_data[1].valid := 1, [1197].log_data[2].valid := 1, [1197].log_data[3].valid := 1, [1197].log_data[4].valid := 1, [1197].log_data[5].valid := 1, [1197].log_data[6].valid := 1, [1197].log_data[7].valid := 1, [1197].log_data[8].valid := 1, [1197].log_data[9].valid := 1, [1197].log_data[10].valid := 1, [1197].log_data[11].valid := 1, [1197].log_data[12].valid := 1, [1197].log_data[13].valid := 1, [1197].log_data[14].valid := 1, [1197].log_data[15].valid := 1, [1197].log_data[16].valid := 1, [1197].log_data[17].valid := 1, [1197].log_data[18].valid := 1, [1197].log_data[19].valid := 1, [1197].time.Year := 2023, [1197].time.Month := 1, [1197].time.Day := 13, [1197].time.Hour := 20, [1197].time.Minute := 9, [1197].time.Second := 59, [1198].log_data[0].min := 1.0, [1198].log_data[0].max := 1.0, [1198].log_data[0].total := 300.0, [1198].log_data[0].time := 300.0, [1198].log_data[0].minminute := 10, [1198].log_data[0].maxminute := 10, [1198].log_data[0].valid := 1, [1198].log_data[1].valid := 1, [1198].log_data[2].valid := 1, [1198].log_data[3].valid := 1, [1198].log_data[4].valid := 1, [1198].log_data[5].valid := 1, [1198].log_data[6].valid := 1, [1198].log_data[7].valid := 1,
